# B&R Automation Studio project VisionSample (part 9)

#### Main.st
```iecst
// -----------------------------------------------------------------------------------------------------------
// Use this task to add your own code
// -----------------------------------------------------------------------------------------------------------

// -----------------------------------------------------------------------------------------------------------
// Initialization
// -----------------------------------------------------------------------------------------------------------
PROGRAM _INIT
	cmdLoadRecipeAfterBoot	:= TRUE;
END_PROGRAM

// -----------------------------------------------------------------------------------------------------------
// Cyclic part
// -----------------------------------------------------------------------------------------------------------
PROGRAM _CYCLIC
		// -----------------------------------------------------------------------------------------------------------
	// Vision sensor configuration
	// -----------------------------------------------------------------------------------------------------------
	gVisionImage.CFG.EthDevice				:= 'IF2';			// Ethernet interface for the PLC, this is the IF where you go online
	// Configuration for blob
	gVisionSensor[1].CFG.VisionFunction		:= enumBlob;		// Used to run specific code for this vision function
	gVisionSensor[1].CFG.PowerlinkNode		:= 1;				// Powerlink node number
	gVisionSensor[1].CFG.DataStructure		:= ADR(gBlob);		// Global structures that holds all data related to this function
	gVisionSensor[1].CFG.ComponentLink		:= gCameraBlob;		// Vision component name defined under mappVision in the configuration view
	gVisionSensor[1].CFG.ResolutionWidth_X	:= 1280;
	gVisionSensor[1].CFG.ResolutionHeight_Y	:= 1024;
	// Configuration for code reader
	gVisionSensor[2].CFG.VisionFunction		:= enumCoderReader;
	gVisionSensor[2].CFG.PowerlinkNode		:= 2;
	gVisionSensor[2].CFG.DataStructure		:= ADR(gCodeReader);
	gVisionSensor[2].CFG.ComponentLink		:= gCameraCodeReading;
	gVisionSensor[2].CFG.ResolutionWidth_X	:= 1280;
	gVisionSensor[2].CFG.ResolutionHeight_Y	:= 1024;
	// Configuration for match
	gVisionSensor[3].CFG.VisionFunction		:= enumMatch;
	gVisionSensor[3].CFG.PowerlinkNode		:= 3;
	gVisionSensor[3].CFG.DataStructure		:= ADR(gMatch);
	gVisionSensor[3].CFG.ComponentLink		:= gCameraMatch;
	gVisionSensor[3].CFG.ResolutionWidth_X	:= 1280;
	gVisionSensor[3].CFG.ResolutionHeight_Y	:= 1024;
	// Configuration for meaurement
	gVisionSensor[4].CFG.VisionFunction		:= enumMeasurement;
	gVisionSensor[4].CFG.PowerlinkNode		:= 4;
	gVisionSensor[4].CFG.DataStructure		:= ADR(gMT);
	gVisionSensor[4].CFG.ComponentLink		:= gCameraMeasurement;
	gVisionSensor[4].CFG.ResolutionWidth_X	:= 1280;
	gVisionSensor[4].CFG.ResolutionHeight_Y	:= 1024;
	// Configuration for OCR
	gVisionSensor[5].CFG.VisionFunction		:= enumOCR;
	gVisionSensor[5].CFG.PowerlinkNode		:= 5;
	gVisionSensor[5].CFG.DataStructure		:= ADR(gOCR);
	gVisionSensor[5].CFG.ComponentLink		:= gCameraOCR;
	gVisionSensor[5].CFG.ResolutionWidth_X	:= 1280;
	gVisionSensor[5].CFG.ResolutionHeight_Y	:= 1024;
	// Configuration for PixelCounter
	gVisionSensor[6].CFG.VisionFunction		:= enumPixelCounter;
	gVisionSensor[6].CFG.PowerlinkNode		:= 6;
	gVisionSensor[6].CFG.DataStructure		:= ADR(gPixel);
	gVisionSensor[6].CFG.ComponentLink		:= gCameraPxl;
	gVisionSensor[6].CFG.ResolutionWidth_X	:= 1280;
	gVisionSensor[6].CFG.ResolutionHeight_Y	:= 1024;

	// -----------------------------------------------------------------------------------------------------------
	// Lights configuration
	// -----------------------------------------------------------------------------------------------------------
	// Configuration for backlights
	gVisionLight[1].CFG.LightType		:= enumBacklight;
	gVisionLight[1].CFG.PowerlinkNode	:= 10;
	gVisionLight[1].DAT.FlashColor		:= 1;
	gVisionLight[2].CFG.LightType		:= enumBacklight;
	gVisionLight[2].CFG.PowerlinkNode	:= 11;
	gVisionLight[2].DAT.FlashColor		:= 1;
	// Configuration for lightbars
	gVisionLight[3].CFG.LightType		:= enumLightbar;
	gVisionLight[3].CFG.PowerlinkNode	:= 20;
	gVisionLight[3].DAT.FlashColor		:= 1;

	// -----------------------------------------------------------------------------------------------------------
	// Backlight handling, this block can be deleted when no backlights are used
	// -----------------------------------------------------------------------------------------------------------

	// -----------------------------------------------------------------------------------------------------------
	// Trigger selected backlight when selected sensor is triggered
	IF(EDGEPOS(gVisionSensor[gSelectedSensor].CMD.ImageTrigger)) THEN
		gVisionLight[gSelectedLight].DAT.Exposure		:= gVisionSensor[gSelectedSensor].DAT.Exposure;
		gVisionLight[gSelectedLight].DAT.NettimeDelay	:= gVisionSensor[gSelectedSensor].DAT.NettimeDelay;
		gVisionLight[gSelectedLight].CMD.FlashTrigger	:= TRUE;
	END_IF

	// -----------------------------------------------------------------------------------------------------------
	// Recipe handling, this block can be deleted when no recipes are used
	// -----------------------------------------------------------------------------------------------------------

	// -----------------------------------------------------------------------------------------------------------
	// Transfer data when loading a recipe
	IF EDGENEG(Recipe_01.CMD.Load) OR cmdLoadRecipeAfterBoot THEN
		cmdLoadRecipeAfterBoot := FALSE;
		FOR i := 1 TO MAX_NUM_CAMS DO
			gVisionSensor[i].FCT.ApplicationName	:= RecipeData.Cam[i].ApplicationName;
			gVisionSensor[i].DAT.Exposure			:= RecipeData.Cam[i].Exposure;
			gVisionSensor[i].DAT.FlashColor			:= RecipeData.Cam[i].FlashColor;
			gVisionSensor[i].DAT.FlashSegment		:= RecipeData.Cam[i].FlashSegment;
			gVisionSensor[i].DAT.Focus				:= RecipeData.Cam[i].Focus;
			gVisionSensor[i].DAT.Gain				:= RecipeData.Cam[i].Gain;
			gVisionSensor[i].DAT.MaxItemCnt			:= RecipeData.Cam[i].MaxItemCnt;
			gVisionSensor[i].DAT.Timeout			:= RecipeData.Cam[i].Timeout;
		END_FOR
		FOR i := 1 TO MAX_NUM_LIGHTS DO
			gVisionLight[i].DAT.Exposure			:= RecipeData.Light[i].Exposure;
			gVisionLight[i].DAT.FlashColor			:= RecipeData.Light[i].FlashColor;
			gVisionLight[i].DAT.FlashSegment		:= RecipeData.Light[i].FlashSegment;
			gVisionLight[i].DAT.SetAngle			:= RecipeData.Light[i].SetAngle;
			gVisionLight[i].DAT.Timeout				:= RecipeData.Light[i].Timeout;
		END_FOR
		// Switch vision application when recipe for blob was loaded
		gVisionSensor[1].CMD.VaSwitchApplication := TRUE;
	END_IF

	// -----------------------------------------------------------------------------------------------------------
	// Transfer data cyclic to the remanent variable
	IF NOT Recipe_01.CMD.Load THEN
		FOR i := 1 TO MAX_NUM_CAMS DO
			RecipeData.Cam[i].ApplicationName	:= gVisionSensor[i].FCT.ApplicationName;
			RecipeData.Cam[i].Exposure			:= gVisionSensor[i].DAT.Exposure;
			RecipeData.Cam[i].FlashColor		:= gVisionSensor[i].DAT.FlashColor;
			RecipeData.Cam[i].FlashSegment		:= gVisionSensor[i].DAT.FlashSegment;
			RecipeData.Cam[i].Focus				:= gVisionSensor[i].DAT.Focus;
			RecipeData.Cam[i].Gain				:= gVisionSensor[i].DAT.Gain;
			RecipeData.Cam[i].MaxItemCnt		:= gVisionSensor[i].DAT.MaxItemCnt;
			RecipeData.Cam[i].Timeout			:= gVisionSensor[i].DAT.Timeout;
		END_FOR
		FOR i := 1 TO MAX_NUM_LIGHTS DO
			RecipeData.Light[i].Exposure		:= gVisionLight[i].DAT.Exposure;
			RecipeData.Light[i].FlashColor		:= gVisionLight[i].DAT.FlashColor;
			RecipeData.Light[i].FlashSegment	:= gVisionLight[i].DAT.FlashSegment;
			RecipeData.Light[i].SetAngle		:= gVisionLight[i].DAT.SetAngle;
			RecipeData.Light[i].Timeout			:= gVisionLight[i].DAT.Timeout;
		END_FOR
	END_IF
	IF visSaveRecipe OR visNewRecipe THEN
		IF(visNewRecipe) THEN
			Recipe_01.CMD.New := TRUE;
		ELSE
			Recipe_01.CMD.Save := TRUE;
		END_IF
		visNewRecipe := FALSE;
		visSaveRecipe := FALSE;
	END_IF
END_PROGRAM
```

### Package Logical/Programs/Axis - Program that handles motion axis related tasks

### Program Logical/Programs/Axis/Axis

#### Types.typ
```iecst
TYPE
	hmi_out_typ : 	STRUCT
		positon : REAL;
		veleocity : REAL;
		inVelocity : BOOL;
		inPostion : BOOL;
		powerlinkCycle_us : DINT;
		triggerPosDelta : REAL;
		triggerTimeDelta : DINT; (*In us*)
	END_STRUCT;
	recipe_typ : 	STRUCT
		acceleration : REAL := 360;
		velocity : REAL := 36000;
		axisPositionDelayCycles : REAL;
		visionPreTriggerCycles : REAL;
		axisPositionTrigger : REAL;
		axisPeriod : REAL;
	END_STRUCT;
	hmi_in_cmd_typ : 	STRUCT
		moveAbs : BOOL;
		home : BOOL;
		power : BOOL;
		run : BOOL;
		errReset : BOOL;
	END_STRUCT;
	hmi_in_typ : 	STRUCT
		recipe : recipe_typ;
		cmd : hmi_in_cmd_typ;
	END_STRUCT;
	hmi_typ : 	STRUCT
		in : hmi_in_typ;
		out : hmi_out_typ;
	END_STRUCT;
	local_typ : 	STRUCT
		mpAxisBasic_0 : MpAxisBasic;
		mpAxisBasicPar_0 : MpAxisBasicParType;
		nettimeLastCycle_us : DINT;
		powerlinkCycle_us : DINT;
		axisPositionNow : REAL;
		triggerPosDelta : REAL;
		triggerTimeDelta : DINT; (*In us*)
		mpRecipeRegVar : MpRecipeRegParSync;
	END_STRUCT;
	hw_in_typ : 	STRUCT
		nettime : DINT;
	END_STRUCT;
	hw_typ : 	STRUCT
		in : hw_in_typ;
	END_STRUCT;
END_TYPE
```

#### Main.st
```iecst
// --------------------------------------------------------------------------------------------------------------------
// Motion sample for using nettime
// --------------------------------------------------------------------------------------------------------------------
PROGRAM _INIT
	this.mpAxisBasic_0.Enable			:= TRUE;
	this.mpAxisBasic_0.MpLink			:= ADR(gAxis_1);
	this.mpAxisBasic_0.Parameters		:= ADR(this.mpAxisBasicPar_0);
	this.mpAxisBasic_0();
	this.mpAxisBasicPar_0.Homing.Mode	:= mcHOMING_DEFAULT;

	hmi.in.recipe.axisPeriod				:= 360; // Needs also to be set in the axis configuration
	hmi.in.recipe.axisPositionTrigger		:= 0;
	hmi.in.recipe.axisPositionDelayCycles	:= 1; 	// Number of PLK cycles which the axis position is old when it comes to this task (Time from encoder to now in this task)
	hmi.in.recipe.visionPreTriggerCycles	:= 4; 	// Number of powerlink cycles the trigger has to be send ahead
	// For camera only 4 is good value, for backlight use 12 with a 800us Powerlink cylce

END_PROGRAM

// -----------------------------------------------------------------------------------------------------------
// Cyclic part
// -----------------------------------------------------------------------------------------------------------
PROGRAM _CYCLIC

// -----------------------------------------------------------------------------------------------------------
// Mapp Motion Axis control
// -----------------------------------------------------------------------------------------------------------
	this.mpAxisBasic_0.Power				:= this.mpAxisBasic_0.Active AND this.mpAxisBasic_0.Info.ReadyToPowerOn AND hmi.in.cmd.power;
	this.mpAxisBasic_0.ErrorReset			:= hmi.in.cmd.errReset;
	this.mpAxisBasic_0.Home					:= this.mpAxisBasic_0.PowerOn AND NOT this.mpAxisBasic_0.IsHomed XOR hmi.in.cmd.home;
	this.mpAxisBasic_0.MoveVelocity			:= this.mpAxisBasic_0.PowerOn AND this.mpAxisBasic_0.IsHomed AND hmi.in.cmd.run;

	IF this.mpAxisBasic_0.PowerOn AND this.mpAxisBasic_0.IsHomed AND hmi.in.cmd.moveAbs THEN
		this.mpAxisBasic_0.MoveAbsolute		:= TRUE;
		this.mpAxisBasicPar_0.Position		:= hmi.in.recipe.axisPositionTrigger;
	END_IF
	hmi.in.cmd.moveAbs					:= FALSE;

	IF hmi.in.recipe.velocity <> this.mpAxisBasicPar_0.Velocity OR hmi.in.recipe.acceleration <> this.mpAxisBasicPar_0.Acceleration THEN
		this.mpAxisBasicPar_0.Velocity		:= hmi.in.recipe.velocity;
		this.mpAxisBasicPar_0.Acceleration	:= hmi.in.recipe.acceleration;
		this.mpAxisBasicPar_0.Deceleration	:= hmi.in.recipe.acceleration;
		this.mpAxisBasic_0.Update			:= TRUE;
	END_IF

	this.mpAxisBasic_0();

	IF hw.in.nettime > this.nettimeLastCycle_us THEN
		this.powerlinkCycle_us	:= hw.in.nettime - this.nettimeLastCycle_us;
	ELSE
		this.powerlinkCycle_us	:= -2147483648-hw.in.nettime + 2147483647-this.nettimeLastCycle_us; // handle wrap around
	END_IF
	this.nettimeLastCycle_us		:= hw.in.nettime;

	hmi.out.inVelocity 	:= gAxis.status.inVelocity	:= 	this.mpAxisBasic_0.InVelocity;
	hmi.out.veleocity 	:= gAxis.status.velocity	:= 	this.mpAxisBasic_0.Velocity;
	hmi.out.inPostion 								:=	this.mpAxisBasic_0.InPosition;
	// When the MpAxis gives us the read position, it is old. So calculate the "now" position
	hmi.out.positon 	:= gAxis.status.position	:= 	LREAL_TO_REAL(this.mpAxisBasic_0.Position) + this.mpAxisBasic_0.Velocity * DINT_TO_REAL(this.powerlinkCycle_us) * hmi.in.recipe.axisPositionDelayCycles / 1000000; ;

	IF this.mpAxisBasic_0.UpdateDone THEN
		this.mpAxisBasic_0.Update := FALSE;
	END_IF

	IF this.mpAxisBasic_0.InPosition THEN
		this.mpAxisBasic_0.MoveAbsolute		:= FALSE;
	END_IF

	// -----------------------------------------------------------------------------------------------------------
	// Calulate time to camera trigger point
	// -----------------------------------------------------------------------------------------------------------

	// calculate axis postion in the current period
	IF this.axisPositionNow > hmi.in.recipe.axisPeriod THEN // modulo correction
		this.axisPositionNow		:= hmi.out.positon- hmi.in.recipe.axisPeriod;
	ELSIF this.axisPositionNow < 0 THEN // modulo correction
		this.axisPositionNow		:= hmi.out.positon + hmi.in.recipe.axisPeriod;
	END_IF

	// calculate differen (triggerPosDelta) in current axis postion to the trigger postion
	IF this.mpAxisBasic_0.Velocity > 0 THEN
		this.triggerPosDelta		:= hmi.in.recipe.axisPositionTrigger - this.axisPositionNow;
	ELSE
		this.triggerPosDelta		:= this.axisPositionNow - hmi.in.recipe.axisPositionTrigger;
	END_IF

	IF this.triggerPosDelta < 0 THEN // modulo correction
		this.triggerPosDelta		:= this.triggerPosDelta + hmi.in.recipe.axisPositionTrigger;
	END_IF

	IF hmi.out.veleocity > 0 THEN
		// convert position difference to a time difference (the time until the axis is at the trigger postion with the current velocity)
		gAxis.status.triggerTimeDelta 	:= LREAL_TO_DINT((this.triggerPosDelta / this.mpAxisBasic_0.Velocity) * 1000000);
	END_IF

	gAxis.status.nettime 		  		:= hw.in.nettime;
	gAxis.status.powerlinkCycleTime 	:= this.powerlinkCycle_us;

	hmi.out.triggerPosDelta 	:= this.triggerPosDelta;
	hmi.out.powerlinkCycle_us 	:= this.powerlinkCycle_us;
	hmi.out.triggerTimeDelta 	:= this.triggerTimeDelta;

	this.mpRecipeRegVar.Enable 		:= gRecipe.out.active;
	this.mpRecipeRegVar.MpLink 		:= gRecipe.out.mpLink;
	this.mpRecipeRegVar.ConfirmSave := this.mpRecipeRegVar.SaveNotification;
	this.mpRecipeRegVar.Category 	:= ADR('Recipe');
	this.mpRecipeRegVar.PVName 		:= ADR('::Axis:hmi.in.recipe');
	this.mpRecipeRegVar();

	// Clear ready for init (auto load) if data structures have not been registred
	IF NOT this.mpRecipeRegVar.Active THEN
		gRecipe.in.readyForInit := FALSE;
	END_IF

END_PROGRAM
```

### Package Logical/Programs/Files - Program that handles file system tasks

### gFiles.typ
```iecst
TYPE
	gFiles_input_typ : 	STRUCT
		refresh : BOOL;
	END_STRUCT;
	gFiles_output_typ : 	STRUCT
		fileDevice : STRING[10];
		ready : BOOL;
	END_STRUCT;
	gFiles_typ : 	STRUCT
		output : gFiles_output_typ;
		input : gFiles_input_typ;
	END_STRUCT;
END_TYPE
```

### Program Logical/Programs/Files/Files

#### Types.typ
```iecst
TYPE
	local_typ : 	STRUCT
		brdkFileDevUsb : brdkFileDeviceHandler;
		brdkFileDev : brdkFileDeviceHandler;
		mpFileManUI : MpFileManagerUI;
		mpFileUISetup : MpFileManagerUISetupType;
		mappView : brdkViImg_mappView;
		lastFileName : STRING[255];
		brdkFileRead : brdkFileRead;
		fileName : STRING[255];
		fileType : STRING[5];
		delayTon : TON;
		setIdx : BOOL;
	END_STRUCT;
	hmi_in_cmd_typ : 	STRUCT
		deleteAllImages : BOOL;
		selectedIdx : UINT;
		download : BOOL;
	END_STRUCT;
	hmi_in_typ : 	STRUCT
		cmd : hmi_in_cmd_typ;
	END_STRUCT;
	hmi_out_typ : 	STRUCT
		enableDeleteAllImageBtn : BOOL;
		fileNames : ARRAY[0..FILES_LIST_SIZE]OF STRING[255];
		loadFileStatus : STRING[200];
		img : STRING[8000000];
		svg : STRING[1000000];
		downloadSrc : STRING[500];
	END_STRUCT;
	hmi_typ : 	STRUCT
		in : hmi_in_typ;
		out : hmi_out_typ;
		mpFile : MpFileManagerUIConnectType;
	END_STRUCT;
END_TYPE
```

#### Variables.var
```iecst
VAR CONSTANT
	FILES_LIST_SIZE : USINT := 13; (*Number of files to be displayed on one page of the list in the HMI application*)
END_VAR
VAR
	hmi : hmi_typ;
	i : UINT;
	this : local_typ;
END_VAR
```

#### Main.st
```iecst
PROGRAM _INIT
	(* Insert code here *)
	this.brdkFileDev.enable := TRUE;
	this.brdkFileDev.setup.plcDrive := F_DRIVE;
	this.brdkFileDev.setup.usbOverrule := FALSE;
	this.brdkFileDev.simulation.pcRootFolder := 'plcSim\MappVisionDemo';
	this.brdkFileDev.simulation.pcHDDrive := C_DRIVE;
	this.brdkFileDev.setup.rootFileDeviceName := 'ROOT_PLC';

	this.brdkFileDev.setup.fileDevices[0].name := 'SIM_BLOB';
	this.brdkFileDev.setup.fileDevices[0].path := 'sim/BLOB';
	this.brdkFileDev.setup.fileDevices[1].name := 'SIM_CR';
	this.brdkFileDev.setup.fileDevices[1].path := 'sim/CR';
	this.brdkFileDev.setup.fileDevices[2].name := 'SIM_MATCH';
	this.brdkFileDev.setup.fileDevices[2].path := 'sim/Match';
	this.brdkFileDev.setup.fileDevices[3].name := 'SIM_MEAS';
	this.brdkFileDev.setup.fileDevices[3].path := 'sim/Measurement';
	this.brdkFileDev.setup.fileDevices[4].name := 'SIM_OCR';
	this.brdkFileDev.setup.fileDevices[4].path := 'sim/OCR';
	this.brdkFileDev.setup.fileDevices[5].name := 'SIM_PXCNT';
	this.brdkFileDev.setup.fileDevices[5].path := 'sim/PxCnt';

	this.brdkFileDevUsb.setup.plcDrive := F_DRIVE;
	this.brdkFileDevUsb.setup.usbOverrule := TRUE;
	this.brdkFileDevUsb.simulation.pcRootFolder := 'plcSim\MappVisionDemo';
	this.brdkFileDevUsb.simulation.pcHDDrive := C_DRIVE;
	this.brdkFileDevUsb.simulation.pcUSBDrive := D_DRIVE;
	this.brdkFileDevUsb.setup.rootFileDeviceName := 'ROOT_USB';

	this.brdkFileDevUsb.setup.fileDevices[0].name := 'IMG';
	this.brdkFileDevUsb.setup.fileDevices[0].path := 'images';
	this.brdkFileDevUsb.setup.fileDevices[1].name := 'RECIPE';
	this.brdkFileDevUsb.setup.fileDevices[1].path := 'Recipe';
	this.brdkFileDevUsb.setup.fileDevices[2].name := 'VI_DIAG';
	this.brdkFileDevUsb.setup.fileDevices[2].path := 'visionDiag';
	this.brdkFileDevUsb.setup.fileDevices[3].name := 'DATA';
	this.brdkFileDevUsb.setup.fileDevices[3].path := 'data';

	this.mpFileManUI.UISetup.FileListScrollWindow := 1;
	this.mpFileManUI.UISetup.FileListSize := FILES_LIST_SIZE;

	this.mappView.simulateConfig.activate := TRUE;
	this.mappView.simulateConfig.appendNumber := FALSE;
	this.mappView.simulateConfig.autoIncrementNumber := FALSE;
	this.mappView.simulateConfig.pDevice := ADR('IMG');
	this.mappView.simulateConfig.useRandomNumbers := FALSE;

	hmi.mpFile.File.Filter := '*jpg';

END_PROGRAM

PROGRAM _CYCLIC
	(* Insert code here *)

	// Create file devices
	this.brdkFileDev();

	IF EDGEPOS(this.brdkFileDev.ready) THEN
		this.brdkFileDevUsb.enable := TRUE;
	END_IF

	hmi.mpFile.File.Refresh := hmi.mpFile.File.Refresh OR gFiles.input.refresh;
	gFiles.input.refresh := FALSE;
	this.brdkFileDevUsb();

	gFiles.output.fileDevice := 'ROOT';
	gFiles.output.ready := this.brdkFileDevUsb.ready;

	// Use MpFile to handle the images files
	hmi.mpFile.DeviceList.DeviceNames[0] := 'IMG';

	this.mpFileManUI.Enable := this.brdkFileDevUsb.ready;
	this.mpFileManUI.MpLink := ADR(gFileManagerUI);
	this.mpFileManUI.UIConnect := ADR(hmi.mpFile);
	IF hmi.mpFile.File.List.PageDown OR hmi.mpFile.File.List.PageUp OR hmi.mpFile.File.List.StepDown OR hmi.mpFile.File.List.StepUp THEN
		this.setIdx := TRUE;
	END_IF

	IF NOT hmi.mpFile.File.List.Items[hmi.in.cmd.selectedIdx].IsSelected THEN
		IF this.setIdx THEN
			this.setIdx := FALSE;
		ELSE

			FOR i := 0 TO this.mpFileManUI.UISetup.FileListSize BY 1 DO
				hmi.mpFile.File.List.Items[i].IsSelected := i = hmi.in.cmd.selectedIdx;
			END_FOR
		END_IF

	END_IF

	this.mpFileManUI();

	FOR i:= 0 TO this.mpFileManUI.UISetup.FileListSize BY 1 DO
		hmi.out.fileNames[i] := hmi.mpFile.File.List.Items[i].Name;
	END_FOR

	IF this.setIdx THEN
		FOR i := 0 TO this.mpFileManUI.UISetup.FileListSize BY 1 DO
			IF hmi.mpFile.File.List.Items[i].IsSelected THEN
				hmi.in.cmd.selectedIdx := i;
			END_IF
		END_FOR
	END_IF

	// Load image and overlay when the selected image changes.
	IF hmi.mpFile.File.List.Items[hmi.in.cmd.selectedIdx].Name <> this.lastFileName THEN
		this.fileName := hmi.mpFile.File.List.Items[hmi.in.cmd.selectedIdx].Name;
		brsstrcpy(ADR(this.fileType),ADR(this.fileName)+brsstrlen(ADR(this.fileName))-3);

		brsstrcpy(ADR(this.fileName)+brsstrlen(ADR(this.fileName))-4,ADR(''));
		this.mappView.simulateConfig.pFile := ADR(this.fileName);

		IF this.fileType = 'jpg' THEN
			this.mappView.imageFormat := BRDKVIIMG_IMG_TYPE_JPEG;
		ELSE
			this.mappView.imageFormat := BRDKVIIMG_IMG_TYPE_BMP;
		END_IF

		this.mappView.updateImage := TRUE;
		this.brdkFileRead.enable := TRUE;

		this.brdkFileRead.fileDevice := hmi.mpFile.DeviceList.DeviceNames[hmi.mpFile.DeviceList.SelectedIndex];
		this.brdkFileRead.fileName := hmi.mpFile.File.List.Items[hmi.in.cmd.selectedIdx].Name;
		brsstrcpy(ADR(this.brdkFileRead.fileName)+brsstrlen(ADR(this.brdkFileRead.fileName))-3,ADR('svg'));
		this.brdkFileRead.pData := ADR(hmi.out.svg);
		this.brdkFileRead.dataLength := SIZEOF(hmi.out.svg);

	END_IF

	this.lastFileName := hmi.mpFile.File.List.Items[hmi.in.cmd.selectedIdx].Name;
	this.brdkFileRead();

	IF this.brdkFileRead.done OR this.brdkFileRead.status = fiERR_FILE_NOT_FOUND THEN
		this.brdkFileRead.enable := FALSE;
	END_IF

	IF hmi.mpFile.MessageBox.Type =  mpFILE_MSG_CONFIRM_DELETE THEN
		hmi.mpFile.MessageBox.Confirm := TRUE;
	END_IF

	IF hmi.in.cmd.download THEN
		hmi.in.cmd.download	:= FALSE;
		this.delayTon.IN 	:= TRUE;
		this.delayTon.PT 	:= T#400ms;

		hmi.out.downloadSrc := '<script>function onSvgLoad() {const link = document.createElement("a");link.href = "/FileDevice:';
		brsstrcat(ADR(hmi.out.downloadSrc),ADR(this.brdkFileRead.fileDevice));
		brsstrcat(ADR(hmi.out.downloadSrc),ADR('/'));
		brsstrcat(ADR(hmi.out.downloadSrc),ADR(hmi.mpFile.File.List.Items[hmi.in.cmd.selectedIdx].Name));
		brsstrcat(ADR(hmi.out.downloadSrc),ADR('";link.download="'));
		brsstrcat(ADR(hmi.out.downloadSrc),ADR(hmi.mpFile.File.List.Items[hmi.in.cmd.selectedIdx].Name));
		brsstrcat(ADR(hmi.out.downloadSrc),ADR('";link.click();}; onSvgLoad(); </script>'));
	END_IF

	IF this.delayTon.Q THEN
		this.delayTon.IN := FALSE;
		hmi.out.downloadSrc := '';
	END_IF
	this.delayTon();

	hmi.out.loadFileStatus := this.brdkFileRead.description;

	this.mappView.enable := this.brdkFileDevUsb.ready;
	this.mappView.wsPort :=  18100;
	//	this.mappView.pSvgImage := ADR(hmi.out.img);
	//	this.mappView.maxSvgImageLength := SIZEOF(hmi.out.img);
	this.mappView();

END_PROGRAM

PROGRAM _EXIT
	(* Insert code here *)
	this.brdkFileDev(	enable := FALSE);
	this.brdkFileDevUsb(enable := FALSE);
	this.mappView(		enable := FALSE);
	this.mpFileManUI(	Enable := FALSE);

END_PROGRAM
```

### Package Logical/Programs/Vision - Main program that handles triggering and processing of vision

### Program Logical/Programs/Vision/Vision (IEC)

#### Main.st - Init, cyclic, exit code
```iecst
// --------------------------------------------------------------------------------------------------------------------
// General vision task. This is a support task for the mappVision. The following functions are implemneted
// - Translate some values in text messages
// - Reset camera trigger when inspection is finsihed
// - Load vision application
// - Save diagnostic data
// Version 2.x (Check revision history for details)
// --------------------------------------------------------------------------------------------------------------------
PROGRAM _INIT

	userInitCommonPreAction;

	FOR idx:= START_IDX TO MAX_NUM_CAMS BY 1 DO
		setupPointersAction;

		//  Create IO path to cam
		this.path := 'IF3.ST';
		tmpStr := USINT_TO_STRING(idx);
		brsstrcat(ADR(this.path),ADR(tmpStr));

		this.recipePVName := '::Vision1:hmiInstance[';
		brsstrcat(ADR(this.recipePVName),ADR(tmpStr));
		brsstrcat(ADR(this.recipePVName),ADR('].in.recipe'));

		// Create IO path to lights
		FOR i := START_IDX TO MAX_NUM_LIGHTS BY 1 DO
			this.lightPath[i] := 'IF3.ST';
			tmpStr := USINT_TO_STRING(idx*16+(i-1));
			brsstrcat(ADR(this.lightPath[i]),ADR(tmpStr));
		END_FOR

		FOR i:= START_IDX TO MAX_NUM_RESULTS BY 1 DO
			hmi.out.tableVF.tableNum[i] := i;
		END_FOR

		hmi.out.wsPort := 18000+idx*10;
		this.mappView.enable := TRUE;
		this.mappView.wsPort := hmi.out.wsPort;
		this.mappView.simulateConfig.activate := DiagCpuIsSimulated();
		this.mappView.simulateConfig.pFile := ADR('img');
		this.mappView.simulateConfig.useRandomNumbers := FALSE;
		this.mappView.simulateConfig.appendNumber := TRUE;
		this.mappView.simulateConfig.autoIncrementNumber := TRUE;
		this.mappView.simulateConfig.minNumber := 1;
		this.mappView.simulateConfig.maxNumber := 3;

		this.visionDiagFileDevice := 'VI_DIAG'; // File device is created in Files program (changes to USB if such is pluged in)

		hmi.out.camera.plNodeNr := idx;
		hmi.in.recipe.cam.focus := 200;
		hmi.in.recipe.cam.exposureTime := 100;

		hmi.in.cmd.resetInfo := TRUE;

		// -----------------------------------------------------------------------------------------------------------
		// Set camera specific data
		// -----------------------------------------------------------------------------------------------------------

		hmi.in.cmd.resultTabIndex := 5;
		CASE idx OF
			1:
				this.mappView.pMappLink := ADR(gCameraBlob);
				this.mappView.simulateConfig.pDevice := ADR('SIM_BLOB');
				hmi.out.camera.visionFunction := 'BLOB';
				hmi.out.usedVF.BLOB := TRUE;
				hmi.in.cmd.resultTabIndex := MIN(hmi.in.cmd.resultTabIndex,idx-1);
			2:
				this.mappView.pMappLink := ADR(gCameraCodeReading);
				this.mappView.simulateConfig.pDevice := ADR('SIM_CR');
				hmi.out.camera.visionFunction := 'Code Reader';
				hmi.out.usedVF.codeReader := TRUE;
				hmi.in.cmd.resultTabIndex := MIN(hmi.in.cmd.resultTabIndex,idx-1);
				(*hmi.out.VF.numResults*)
			3:
				this.mappView.pMappLink := ADR(gCameraMatch);
				this.mappView.simulateConfig.pDevice := ADR('SIM_MATCH');
				hmi.out.camera.visionFunction := 'Matching';
				hmi.out.usedVF.matching := TRUE;
				hmi.in.cmd.resultTabIndex := MIN(hmi.in.cmd.resultTabIndex,idx-1);
			4:
				this.mappView.pMappLink := ADR(gCameraMeasurement);
				this.mappView.simulateConfig.pDevice := ADR('SIM_MEAS');
				hmi.out.camera.visionFunction := 'Measurement';
				hmi.out.usedVF.measurement := TRUE;
				hmi.in.cmd.resultTabIndex := MIN(hmi.in.cmd.resultTabIndex,idx-1);
			5:
				this.mappView.pMappLink := ADR(gCameraOCR);
				this.mappView.simulateConfig.pDevice := ADR('SIM_OCR');
				hmi.out.camera.visionFunction := 'OCR';
				hmi.out.usedVF.OCR := TRUE;
				hmi.in.cmd.resultTabIndex := MIN(hmi.in.cmd.resultTabIndex,idx-1);
			6:
				this.mappView.pMappLink := ADR(gCameraPxl);
				this.mappView.simulateConfig.pDevice := ADR('SIM_PXCNT');
				hmi.out.camera.visionFunction := 'Pixel Counter';
				hmi.out.usedVF.pixelCounter := TRUE;
				hmi.in.cmd.resultTabIndex := MIN(hmi.in.cmd.resultTabIndex,idx-1);

		END_CASE

		userInitLocalPostAction;

	END_FOR

END_PROGRAM

// -----------------------------------------------------------------------------------------------------------
// Cyclic part
// -----------------------------------------------------------------------------------------------------------
PROGRAM _CYCLIC

	userCommonPreAction; // user common action before all other

	FOR idx:= START_IDX TO MAX_NUM_CAMS BY 1 DO
		setupPointersAction;

		userLocalPreAction; // user local action before all other

		// -----------------------------------------------------------------------------------------------------------
		// Translate camera status in readable text
		// -----------------------------------------------------------------------------------------------------------
		IF hw.camera.in.common.moduleOk THEN
			brdkViBase_camStatusToString(hw.camera.in.status.cameraStatus,ADR(hmi.out.camera.statusText));
		ELSE
			hmi.out.camera.statusText := 'Disconnected';
		END_IF

		// -----------------------------------------------------------------------------------------------------------
		// Check if vision cockpit is open
		// -----------------------------------------------------------------------------------------------------------
		hmi.out.camera.mappVisionActive := (hw.camera.in.status.cameraStatus AND 16#8000_0000) > 0;

		// -----------------------------------------------------------------------------------------------------------
		// Read camera hardware info
		// -----------------------------------------------------------------------------------------------------------

		IF hmi.in.cmd.resetInfo THEN
			hmi.in.cmd.resetInfo := FALSE;
			hmi.in.cameraInfo.distance := hmi.in.recipe.cam.focus;
			this.brdkViBase_getCameraInfo_0.execute := TRUE;
			this.brdkViBase_getCameraInfo_0.pluggedModule := hw.camera.in.common.moduleOk AND NOT DiagCpuIsSimulated();

			FOR i := START_IDX TO MAX_NUM_LIGHTS BY 1 DO
				this.brdkViBase_getLightInfo[i].execute := TRUE;
				this.brdkViBase_getLightInfo[i].pInfo := ADR(hmi.out.lights[i].info);
				this.brdkViBase_getLightInfo[i].pDevicePath := ADR(this.lightPath[i]);
				this.brdkViBase_getLightInfo[i].pluggedModule := hw.lights[i].in.common.moduleOk AND NOT DiagCpuIsSimulated();
			END_FOR

		END_IF

		this.brdkViBase_getCameraInfo_0.pDevicePath := ADR(this.path);
		this.brdkViBase_getCameraInfo_0.pInfo := ADR(hmi.in.cameraInfo);
		this.brdkViBase_getCameraInfo_0();

		FOR i:=START_IDX TO MAX_NUM_LIGHTS BY 1 DO
			this.brdkViBase_getLightInfo[i]();

			IF hmi.out.lights[i].info.orderNr <> '' AND this.brdkViBase_getLightInfo[i].status = ERR_OK THEN
				// set Camera flash options based on current camera
				brdkViBase_LEDColorToOptions(hmi.out.lights[i].info.LED_color, ADR(hmi.out.lights[i].flashLightOptions));
			END_IF
		END_FOR

		IF hw.camera.out.par.focus <> hmi.in.recipe.cam.focus THEN
			hmi.in.cameraInfo.distance := hmi.in.recipe.cam.focus;
		END_IF

		IF hmi.in.cameraInfo.orderNr <> '' AND this.brdkViBase_getCameraInfo_0.status = ERR_OK THEN
			brdkViBase_calcOpticInfo(hmi.in.cameraInfo, hmi.out.camera.opticInfo); // calculate optic info based on defined info

			// set Camera flash options based on current camera
			brdkViBase_LEDColorToOptions(hmi.in.cameraInfo.LED_color, ADR(hmi.out.camera.flashLightOptions));
		END_IF

		IF hw.io.in.nettime > this.axisTrig.nettimeLastCycle_us THEN
			this.axisTrig.powerlinkCycle_us	:= hw.io.in.nettime - this.axisTrig.nettimeLastCycle_us;
		ELSE
			this.axisTrig.powerlinkCycle_us	:= -2147483648-hw.io.in.nettime + 2147483647-this.axisTrig.nettimeLastCycle_us; // handle wrap around
		END_IF
		this.axisTrig.nettimeLastCycle_us	:= hw.io.in.nettime;

		// -----------------------------------------------------------------------------------------------------------
		// Image trigger (camera and lights)
		// -----------------------------------------------------------------------------------------------------------
		hmi.in.recipe.cam.flashColor := STRING_TO_USINT(hmi.in.recipe.cam.flashColorStr);
		hw.camera.out.par.focus 			:= hmi.in.recipe.cam.focus;
		hw.camera.out.par.flashSegment	 	:= hmi.in.recipe.cam.flashSegment;
		hw.camera.out.par.flashColor 		:= hmi.in.recipe.cam.flashColor;
		hw.camera.out.par.exposureTime 		:= hmi.in.recipe.cam.exposureTime;
		hw.camera.out.par.chromaticLock 	:= hmi.in.recipe.cam.chromaticLock;
		hw.camera.out.par.gainLevel 		:= hmi.in.recipe.cam.gainLevel;
		hw.camera.out.par.IRFilter			:= hmi.in.recipe.cam.IRFilter;

		//-------------------------------------------------------------------------

		// Copy recipe data (e.g. enable, maximal number of results, etc.)
		hw.VF.blob.out			:=hmi.in.recipe.BLOB;
		hw.VF.codeReader.out	:= hmi.in.recipe.CR;
		hw.VF.matching.out		:=hmi.in.recipe.match;
		hw.VF.measurement.out	:=hmi.in.recipe.meassurement;
		hw.VF.ocr.out			:=hmi.in.recipe.OCR;
		hw.VF.pixelCnt.out		:=hmi.in.recipe.pxCnt;

		hmi.out.camera.processingTime:=hw.camera.in.status.cameraProcessingTime;

		CASE idx OF
			1:
				hmi.out.VF.processingTime := hw.VF.blob.in.common.functionProcessingTime;
				hmi.out.VF.numResults := hw.VF.blob.in.common.numResults;
			2:
				hmi.out.VF.processingTime := hw.VF.codeReader.in.common.functionProcessingTime;
				hmi.out.VF.numResults := hw.VF.codeReader.in.common.numResults;
			3:
				hmi.out.VF.processingTime := hw.VF.matching.in.common.functionProcessingTime;
				hmi.out.VF.numResults := hw.VF.matching.in.common.numResults;
			4:
				hmi.out.VF.processingTime := hw.VF.measurement.in.common.functionProcessingTime;
				hmi.out.VF.numResults := hw.VF.measurement.in.common.numResults;
			5:
				hmi.out.VF.processingTime := hw.VF.ocr.in.common.functionProcessingTime;
				hmi.out.VF.numResults := hw.VF.ocr.in.common.numResults;
			6:
				hmi.out.VF.processingTime := hw.VF.pixelCnt.in.common.functionProcessingTime;
				hmi.out.VF.numResults := hw.VF.pixelCnt.in.common.numResults;
		END_CASE;

		//-------------------------------------------------------------------------

		this.ioTrigger(CLK := hw.io.in.commonTrigger OR hw.io.in.individualTrigger);
		this.repetitiveTriggerTON.IN := hmi.in.recipe.repetitiveTrigger;
		this.repetitiveTriggerTON.PT := UDINT_TO_TIME(hmi.in.recipe.repetitiveTriggerInterval);
		this.repetitiveTriggerTON();

		// check if camera is ready for an image trigger and MappView have been updated
		IF this.brdkViBase_imgTrigger_0.ready AND NOT this.brdkViBase_imgTrigger_0.busy AND this.mappView.status = 0 THEN

			// Hmi manual trigger
			IF hmi.in.cmd.trigger OR this.repetitiveTriggerTON.Q THEN
				hmi.in.cmd.trigger 							:= FALSE;

				this.repetitiveTriggerTON(IN:=FALSE);

				this.brdkViBase_imgTrigger_0.trigger 		:= TRUE;
				this.brdkViBase_imgTrigger_0.delayNettime 	:= hw.io.in.nettime + gAxis.status.powerlinkCycleTime * 12+10000; // Calc nettime close to currnet time
				this.currentTriggerNum := 1;
				// Axis trigger
			ELSIF hmi.in.recipe.enableAxisTrigger AND
				gAxis.status.triggerTimeDelta >= (commonHmi.in.recipe.visionPreTriggerCycles * this.axisTrig.powerlinkCycle_us) AND
				gAxis.status.triggerTimeDelta <= ((commonHmi.in.recipe.visionPreTriggerCycles + 1) * this.axisTrig.powerlinkCycle_us) THEN

				this.brdkViBase_imgTrigger_0.trigger := TRUE;
				this.brdkViBase_imgTrigger_0.delayNettime := gAxis.status.nettime + gAxis.status.triggerTimeDelta; // Use time calculated in Axis program
			ELSIF hmi.in.recipe.enableIoTrigger AND this.ioTrigger.Q THEN

				this.brdkViBase_imgTrigger_0.trigger := TRUE;
				this.brdkViBase_imgTrigger_0.delayNettime := gAxis.status.nettime + hmi.in.recipe.ioTriggerDelay ; // Use time calculated in Axis program

			ELSIF this.currentTriggerNum < hmi.in.recipe.multiCaptureNum AND NOT hmi.in.recipe.repetitiveTrigger THEN

				this.brdkViBase_imgTrigger_0.trigger 		:= TRUE;
				this.brdkViBase_imgTrigger_0.delayNettime 	:= hw.io.in.nettime + gAxis.status.powerlinkCycleTime * 12+10000; // Calc nettime close to currnet time

				this.currentTriggerNum := 		this.currentTriggerNum +1;

			END_IF
		END_IF

		this.brdkViBase_imgTrigger_0.searchAcquisitonSettings := hmi.in.cmd.autoSearch;
		this.brdkViBase_imgTrigger_0.pCameraHw := ADR(hw.camera);
		this.brdkViBase_imgTrigger_0.numLights := MAX_NUM_LIGHTS;
		this.brdkViBase_imgTrigger_0.pLightHw := ADR(hw.lights);
		this.brdkViBase_imgTrigger_0.useCamColorForLight := hmi.in.recipe.useCamLedColorForLight;
		this.brdkViBase_imgTrigger_0.useCamExpTimeForLight := hmi.in.recipe.useCamExpTimeForLight;
		this.brdkViBase_imgTrigger_0.simulate.enable := DiagCpuIsSimulated();
		this.brdkViBase_imgTrigger_0.simulate.alwaysSimulateNonePresentLights := TRUE;
		this.brdkViBase_imgTrigger_0.simulate.imgProcessingDelay := T#300ms;
		this.brdkViBase_imgTrigger_0();

		FOR i:=START_IDX TO MAX_NUM_LIGHTS BY 1 DO

			// Manual Light trigger
			// exposuretime
			IF hmi.in.recipe.useCamExpTimeForLight THEN
				hw.lights[i].out.par.exposureTime := hmi.in.recipe.cam.exposureTime;
			ELSE
				hw.lights[i].out.par.exposureTime := hmi.in.recipe.lights[i].exposureTime;
			END_IF
			// color
			IF hmi.in.recipe.useCamLedColorForLight THEN
				hw.lights[i].out.par.flashColor := hmi.in.recipe.cam.flashColor;
			ELSE
				hw.lights[i].out.par.flashColor := hmi.in.recipe.lights[i].flashColor;
			END_IF

			hmi.out.lights[i].common:=hw.lights[i].in.common;
			hmi.out.lights[i].status:=hw.lights[i].in.status;
			hw.lights[i].out.par.flashAngle:=hmi.in.recipe.lights[i].flashAngle;

			hmi.out.lights[i].plNodeNr := idx*16+UINT_TO_USINT(i-1);

			IF hmi.in.cmd.lights[i].flashTrigger AND NOT hw.lights[i].out.cmd.flashTrigger THEN
				hmi.in.cmd.lights[i].flashTrigger := FALSE;
				hw.lights[i].out.cmd.flashTrigger := TRUE;

				// Nettime
				hw.lights[i].out.par.nettime := hw.io.in.nettime + gAxis.status.powerlinkCycleTime * commonHmi.in.recipe.visionPreTriggerCycles;
			ELSIF 	hw.lights[i].out.cmd.flashTrigger AND hw.lights[i].out.par.nettime <= hw.io.in.nettime THEN
				hw.lights[i].out.cmd.flashTrigger := FALSE;
			END_IF
		END_FOR

		// -----------------------------------------------------------------------------------------------------------
		// New image ready and results
		// -----------------------------------------------------------------------------------------------------------
		// New image (hight for one scan)
		IF this.brdkViBase_imgTrigger_0.newImage THEN

			this.mappView.updateImage := NOT hmi.in.recipe.showOnlyLastImage OR this.currentTriggerNum = hmi.in.recipe.multiCaptureNum; // Trigger an update of the image on hmi
			this.DTGetTime_0(enable := TRUE);

			processResultsAction; // Process results action

			userResultProcessingAction; // User defined process results

		END_IF

		// -----------------------------------------------------------------------------------------------------------
		// Selection of specific result
		// -----------------------------------------------------------------------------------------------------------
		IF hmi.in.cmd.click THEN
			hmi.in.cmd.click := FALSE;

			//VF
			brdkStrSubStr(ADR(tmpVF),ADR(hmi.in.cmd.elemId),1,1);
			//ID
			brsstrcpy(ADR(tmpID),ADR(hmi.in.cmd.elemId)+2);

			hmi.in.cmd.intElemId := STRING_TO_USINT(tmpID);
			IF hmi.in.cmd.intElemId > MAX_NUM_RESULTS THEN
				hmi.in.cmd.intElemId := 0;
			END_IF

		END_IF

		IF hmi.in.cmd.intElemId <> this.oldIntElemID THEN
			this.oldIntElemID := hmi.in.cmd.intElemId;
			processResultsAction;
		END_IF

		// -----------------------------------------------------------------------------------------------------------
		// Auto search vision acquistion settings done (save found settings in recipe structure)
		// -----------------------------------------------------------------------------------------------------------

		// search Auto Focus done (hight for one scan)
		IF this.brdkViBase_imgTrigger_0.searchAcquisitonSettingsDone THEN
			hmi.in.cmd.autoSearch 			:= FALSE;
			hmi.in.recipe.cam.gainLevel 	:=	 hw.camera.in.status.gainLevel;
			hmi.in.recipe.cam.focus		 	:=	 hw.camera.in.status.focus;
			hmi.in.recipe.cam.exposureTime 	:=	 hw.camera.in.status.exposureTime;
			this.brdkViBase_imgTrigger_0.searchAcquisitonSettings := FALSE;
			hmi.in.cmd.trigger 				:= TRUE;
		END_IF

		// -----------------------------------------------------------------------------------------------------------
		// MappView get image to show om hmi
		// -----------------------------------------------------------------------------------------------------------

		IF DiagCpuIsSimulated() THEN
			this.mappView.imageFormat := BRDKVIIMG_IMG_TYPE_JPEG;
		ELSE
			this.mappView.imageFormat := commonHmi.in.recipe.imageFormat;
		END_IF
		this.mappView.jpegQuality := commonHmi.in.recipe.jpegQuality;
		this.mappView();

		// -----------------------------------------------------------------------------------------------------------
		// Save image to file devive F:/images
		// -----------------------------------------------------------------------------------------------------------
		CASE this.saveState OF
			0:

				IF (hmi.in.cmd.saveImage OR (this.mappView.newSvgReady AND commonHmi.in.recipe.saveAllImages))  AND gFiles.output.ready THEN
					hmi.in.cmd.saveImage := FALSE;

					// create filename with VF name and current date of the image
					brsstrcpy(ADR(this.tmpFileName),ADR(hmi.out.camera.visionFunction));
					brsstrcat(ADR(this.tmpFileName),ADR('-'));
					brdkViBase_dateTimeToString(this.DTGetTime_0.DT1,'%Y-%m-%d-%H-%M-%S',ADR(this.tmpFileName));

					brsstrcpy(ADR(this.brdkFileWrite.fileName),ADR(this.tmpFileName));

					CASE this.mappView.imageFormat OF
						BRDKVIIMG_IMG_TYPE_JPEG:
							brsstrcat(ADR(this.brdkFileWrite.fileName),ADR('.jpg'));
						BRDKVIIMG_IMG_TYPE_BMP:
							brsstrcat(ADR(this.brdkFileWrite.fileName),ADR('.bmp'));
					END_CASE

					this.brdkFileWrite.enable := TRUE;
					this.brdkFileWrite.dataLength := this.mappView.internal.getImage.destLen;
					this.brdkFileWrite.pData := this.mappView.internal.getImage.pDest;
					this.brdkFileWrite.overwrite := TRUE;
					this.brdkFileWrite.fileDevice := 'IMG';

					this.saveState := 10;
				END_IF
			10:

				IF this.brdkFileWrite.done THEN
					gFiles.input.refresh := TRUE;
					this.brdkFileWrite.enable := FALSE;
					this.saveState := 20;
				END_IF

			20:
				brsstrcpy(ADR(this.brdkFileWrite.fileName),ADR(this.tmpFileName));

				brsstrcat(ADR(this.brdkFileWrite.fileName),ADR('.svg'));
				this.brdkFileWrite.enable := TRUE;
				this.brdkFileWrite.dataLength := brsstrlen(ADR(hmi.out.svgOverlay));
				this.brdkFileWrite.pData := ADR(hmi.out.svgOverlay);
				this.brdkFileWrite.overwrite := TRUE;
				this.brdkFileWrite.fileDevice := 'IMG';

				this.saveState := 30;

			30:
				IF this.brdkFileWrite.done THEN
					gFiles.input.refresh := TRUE;
					this.brdkFileWrite.enable := FALSE;
					this.saveState := 0;
				END_IF

		END_CASE

		this.brdkFileWrite();

		// -----------------------------------------------------------------------------------------------------------
		// Save diagnostic data
		// -----------------------------------------------------------------------------------------------------------
		IF hmi.in.cmd.saveDiagnositc AND gFiles.output.ready THEN
			hmi.in.cmd.saveDiagnositc 			:= FALSE;

			// Delete old file first
			this.fileDelete.enable 					:= TRUE;
			this.fileDelete.pDevice 				:= ADR(this.visionDiagFileDevice);
			this.fileDelete.pName 					:= ADR(hmi.in.diagnosticFilename);

			// Upload diagnostic information
			this.viBaseSaveDiagData_0.MpLink 		:= this.mappView.pMappLink;
			this.viBaseSaveDiagData_0.DeviceName 	:= ADR(this.visionDiagFileDevice);
			this.viBaseSaveDiagData_0.FileName 		:= ADR(hmi.in.diagnosticFilename);
			hmi.out.camera.saveDiagStatus 			:= UINT_TO_DINT(ERR_FUB_BUSY);
		END_IF

		// file delete done or error (if file do not exsist)
		IF (this.fileDelete.enable AND this.fileDelete.status = ERR_OK) THEN
			this.fileDelete.enable 				:= FALSE;
			this.viBaseSaveDiagData_0.Execute 	:= TRUE;
		END_IF

		// Done
		IF (this.viBaseSaveDiagData_0.Done) THEN
			hmi.out.camera.saveDiagStatus		:= UINT_TO_DINT(ERR_OK);
			this.viBaseSaveDiagData_0.Execute 	:= FALSE;
		END_IF

		// Error
		IF (NOT this.viBaseSaveDiagData_0.Busy AND this.viBaseSaveDiagData_0.Error) THEN
			hmi.out.camera.saveDiagStatus		:= this.viBaseSaveDiagData_0.StatusID;
			this.viBaseSaveDiagData_0.Execute 	:= FALSE;
		END_IF

		this.viBaseSaveDiagData_0();
		this.fileDelete();

		// -----------------------------------------------------------------------------------------------------------
		// Get Vision application list from camera
		// -----------------------------------------------------------------------------------------------------------

		// trigger
		IF hmi.in.cmd.vaList.refresh THEN
			hmi.in.cmd.vaList.refresh 	:= FALSE;

			this.getVaList.Execute 		:= TRUE;
			this.getVaList.Format 		:= viBASE_FORMAT_PLAIN_TEXT;
			this.getVaList.List 		:= ADR(hmi.out.vaList.list);
			this.getVaList.ListLen 		:= SIZEOF(hmi.out.vaList.list);
			this.getVaList.MpLink 		:= this.mappView.pMappLink;
		END_IF

		// Done
		IF this.getVaList.Done THEN
			this.getVaList.Execute 		:= FALSE;
			hmi.out.vaList.length 		:= this.getVaList.NrEntries;
		END_IF

		// Error
		IF this.getVaList.Error THEN
			this.getVaList.Execute 		:= FALSE;
			hmi.out.vaList.lastError 	:= this.getVaList.StatusID;
		END_IF

		this.getVaList();

		// -----------------------------------------------------------------------------------------------------------
		// Load vision application
		// -----------------------------------------------------------------------------------------------------------

		// Trigger
		IF hmi.in.cmd.vaList.load AND brsstrlen(ADR(hmi.out.vaList.list[hmi.in.cmd.vaList.selectedIndex])) > 5 THEN
			hmi.in.cmd.vaList.load 						:= FALSE;

			this.viBaseLoadApplication_0.Execute 	:= TRUE;
			this.viBaseLoadApplication_0.MpLink		:= this.mappView.pMappLink;
			this.viBaseLoadApplication_0.Name		:= ADR(hmi.out.vaList.list[hmi.in.cmd.vaList.selectedIndex]);
			hmi.out.camera.vaLoad 					:= UINT_TO_DINT(ERR_FUB_BUSY);
		ELSE
			hmi.in.cmd.vaList.load := FALSE;
		END_IF

		// Done
		IF (this.viBaseLoadApplication_0.Done) THEN
			hmi.in.cmd.vaList.selectedIndex := 0;
			this.viBaseLoadApplication_0.Execute 	:= FALSE;
			hmi.out.camera.vaLoad 					:= UINT_TO_DINT(ERR_OK);
		END_IF

		// Error
		IF (NOT this.viBaseLoadApplication_0.Busy AND this.viBaseLoadApplication_0.Error) THEN
			this.viBaseLoadApplication_0.Execute 	:= FALSE;
			hmi.out.camera.vaLoad 					:= this.viBaseLoadApplication_0.StatusID;
		END_IF

		this.viBaseLoadApplication_0();

		// -----------------------------------------------------------------------------------------------------------
		// HMI stuff
		// -----------------------------------------------------------------------------------------------------------
		hmiAction;

		// -----------------------------------------------------------------------------------------------------------
		// Recipe handling (register recipse data structure
		// -----------------------------------------------------------------------------------------------------------
		this.mpRecipeRegVar.Enable 		:= gRecipe.out.active;
		this.mpRecipeRegVar.MpLink 		:= gRecipe.out.mpLink;
		this.mpRecipeRegVar.ConfirmSave := this.mpRecipeRegVar.SaveNotification;
		this.mpRecipeRegVar.Category 	:= ADR('Recipe');
		this.mpRecipeRegVar.PVName 		:= ADR(this.recipePVName);
		this.mpRecipeRegVar();

		// handle conversion from CR dropDown value to interger and back
		IF this.mpRecipeRegVar.UpdateNotification THEN
			hmi.in.recipe.CRTypeStr := USINT_TO_STRING(hmi.in.recipe.CR.symbolType);

			FOR i:=START_IDX TO MAX_NUM_LIGHTS BY 1 DO
				this.brdkViBase_getLightInfo[i]();
				hmi.in.cmd.lightColorStr[i] := USINT_TO_STRING(hmi.in.recipe.lights[i].flashColor );
			END_FOR

		ELSE
			hmi.in.recipe.CR.symbolType := STRING_TO_USINT(hmi.in.recipe.CRTypeStr);
			FOR i:=START_IDX TO MAX_NUM_LIGHTS BY 1 DO
				this.brdkViBase_getLightInfo[i]();
				hmi.in.recipe.lights[i].flashColor := STRING_TO_USINT(hmi.in.cmd.lightColorStr[i]);
			END_FOR
		END_IF

		// Clear ready for init (auto load) if data structures have not been registred
		IF NOT this.mpRecipeRegVar.Active THEN
			gRecipe.in.readyForInit := FALSE;
		END_IF

		userLocalPostAction; // user local action after all other

	END_FOR

	userCommonPostAction; // user common action after all other

	// -----------------------------------------------------------------------------------------------------------
	//Configure the pointers (this,hmi,hw etc.) show the correct data for that watch index
	// -----------------------------------------------------------------------------------------------------------
	watchIdx := LIMIT(START_IDX,watchIdx,MAX_NUM_CAMS);
	idx := watchIdx;
	setupPointersAction;

					END_PROGRAM

PROGRAM _EXIT

	FOR idx:= START_IDX TO MAX_NUM_CAMS BY 1 DO
		setupPointersAction;

		this.mappView(enable := FALSE);
		this.mpRecipeRegVar(Enable := FALSE);

		userExitLocalPostAction;
	END_FOR

	userExitCommonPostAction;

					END_PROGRAM
```

#### Types.typ
```iecst
(*Local data structure*)

TYPE
	local_axisTrig_typ : 	STRUCT
		nettimeLastCycle_us : DINT;
		powerlinkCycle_us : DINT;
		axisPositionNow : REAL;
		triggerPosDelta : REAL;
		triggerTimeDelta : DINT; (*In us*)
	END_STRUCT;
	local_vaList_typ : 	STRUCT
	END_STRUCT;
	local_typ : 	STRUCT
		path : STRING[100];
		lightPath : ARRAY[START_IDX..MAX_NUM_LIGHTS]OF STRING[100];
		brdkViBase_imgTrigger_0 : brdkViBase_imgTrigger;
		brdkViBase_getLightInfo : ARRAY[START_IDX..MAX_NUM_LIGHTS]OF brdkViBase_getLightInfo;
		brdkViBase_getCameraInfo_0 : brdkViBase_getCameraInfo;
		mappView : {REDUND_UNREPLICABLE} brdkViImg_mappView;
		viBaseSaveDiagData_0 : ViBaseSaveDiagData;
		fileDelete : FileDelete;
		visionDiagFileDevice : STRING[10];
		viBaseLoadApplication_0 : ViBaseLoadApplication;
		axisTrig : local_axisTrig_typ;
		brdkFileWrite : brdkFileWrite;
		dtNow : DTStructure;
		DTGetTime_0 : DTGetTime;
		tmp2D : brdkViBase_2d_typ;
		strElemId : STRING[80];
		oldIntElemID : USINT;
		elemId : STRING[80];
		tmpAngle : LREAL;
		strStyle : STRING[240];
		mpRecipeRegVar : MpRecipeRegParSync;
		recipePVName : STRING[100];
		getVaList : ViBaseListApplication;
		tmpFileName : STRING[255];
		saveState : USINT;
		ioTrigger : R_TRIG;
		user : user_local_typ;
		currentTriggerNum : UINT;
		repetitiveTriggerTON : TON;
		tmpDraw : hmi_in_recipe_draw_typ;
	END_STRUCT;
END_TYPE

(*Hardware*)

TYPE
	hw_io_in_typ : 	STRUCT
		nettime : DINT;
		commonTrigger : BOOL;
		individualTrigger : BOOL;
	END_STRUCT;
	hw_io_typ : 	STRUCT
		in : hw_io_in_typ;
	END_STRUCT;
	hw_typ : 	STRUCT
		camera : brdkViBase_cam_hw_typ;
		VF : hw_VF_typ;
		lights : ARRAY[START_IDX..MAX_NUM_LIGHTS]OF brdkViBase_light_hw_typ;
		io : hw_io_typ;
		user : user_hw_typ;
	END_STRUCT;
	hw_VF_typ : 	STRUCT
		codeReader : brdkViBase_hw_cr_10_typ;
		pixelCnt : brdkViBase_hw_pxCnt_10_typ;
		measurement : brdkViBase_hw_meas_10_typ;
		matching : brdkViBase_hw_match_10_typ;
		ocr : brdkViBase_hw_OCR_10_typ;
		blob : brdkViBase_hw_blob_10_typ;
	END_STRUCT;
END_TYPE

(*HMI*)

TYPE
	hmi_typ : 	STRUCT
		in : hmi_in_typ;
		out : hmi_out_typ;
		user : user_hmi_typ;
	END_STRUCT;
END_TYPE

(*HMI output*)

TYPE
	hmi_out_typ : 	STRUCT
		svgOverlay : STRING[10000];
		wsPort : UINT;
		lights : ARRAY[START_IDX..MAX_NUM_LIGHTS]OF hmi_out_lights_typ;
		camera : hmi_out_camera_typ;
		VF : hmi_out_vf_typ;
		tableVF : hmi_out_vf_table_typ;
		vaList : hmi_out_vaList_typ;
		usedVF : hmi_out_usedVF_typ;
	END_STRUCT;
	hmi_out_vf_typ : 	STRUCT
		processingTime : UDINT;
		numResults : USINT;
		match : brdkViBase_hmi_match_in_typ;
		measurement : brdkViBase_hw_meas_in_typ;
		codeReader : brdkViBase_hmi_cr_in_typ;
		ocr : brdkViBase_hmi_OCR_in_typ;
		pixelCnt : brdkViBase_hmi_pxCnt_in_typ;
		blob : brdkViBase_hmi_blob_in_typ;
	END_STRUCT;
	hmi_out_lights_typ : 	STRUCT
		status : brdkViBase_light_hw_status_typ;
		common : brdkViBase_hw_in_common_typ;
		simulated : BOOL;
		connectedText : STRING[20];
		connected : BOOL;
		statusText : STRING[50];
		lightType : USINT;
		plNodeNr : USINT;
		info : brdkViBase_lightInfo_typ;
		flashLightOptions : ARRAY[0..4]OF STRING[50];
	END_STRUCT;
	hmi_out_camera_typ : 	STRUCT
		simulated : BOOL;
		connectedText : STRING[20];
		connected : BOOL;
		mappVisionActive : BOOL;
		processing : BOOL;
		ready : BOOL;
		statusText : STRING[50];
		plNodeNr : USINT;
		visionFunction : STRING[20];
		processingTime : UDINT;
		opticInfo : brdkViBase_opticInfo_typ;
		common : brdkViBase_hw_in_common_typ;
		hw : brdkViBase_cam_hw_in_status_typ;
		vaLoad : DINT;
		saveDiagStatus : DINT;
		flashLightOptions : ARRAY[0..4]OF STRING[50];
	END_STRUCT;
	hmi_out_vaList_typ : 	STRUCT
		list : ARRAY[0..99]OF ViBaseFormatPlainTextType;
		length : {REDUND_UNREPLICABLE} UINT;
		lastError : DINT;
	END_STRUCT;
	hmi_out_usedVF_typ : 	STRUCT
		pixelCounter : BOOL;
		measurement : BOOL;
		matching : BOOL;
		codeReader : BOOL;
		OCR : BOOL;
		BLOB : BOOL;
	END_STRUCT;
	hmi_out_vf_table_cr_typ : 	STRUCT  (*Code reader structures*)
		BarcodeText : ARRAY[START_IDX..MAX_NUM_RESULTS]OF STRING[101];
		BarcodeType : ARRAY[START_IDX..MAX_NUM_RESULTS]OF USINT;
		PositionX : ARRAY[START_IDX..MAX_NUM_RESULTS]OF REAL;
		PositionY : ARRAY[START_IDX..MAX_NUM_RESULTS]OF REAL;
		Orientation : ARRAY[START_IDX..MAX_NUM_RESULTS]OF REAL;
		Grading : ARRAY[START_IDX..MAX_NUM_RESULTS]OF SINT;
	END_STRUCT;
	hmi_out_vf_table_blob_typ : 	STRUCT  (*Blob function structures*)
		ModelNumber : ARRAY[START_IDX..MAX_NUM_RESULTS]OF USINT;
		Clipped : ARRAY[START_IDX..MAX_NUM_RESULTS]OF BOOL;
		Area : ARRAY[START_IDX..MAX_NUM_RESULTS]OF REAL;
		PositionX : ARRAY[START_IDX..MAX_NUM_RESULTS]OF REAL;
		PositionY : ARRAY[START_IDX..MAX_NUM_RESULTS]OF REAL;
		Orientation : ARRAY[START_IDX..MAX_NUM_RESULTS]OF REAL;
		MeanGrayValue : ARRAY[START_IDX..MAX_NUM_RESULTS]OF USINT;
		Length : ARRAY[START_IDX..MAX_NUM_RESULTS]OF UDINT;
		Width : ARRAY[START_IDX..MAX_NUM_RESULTS]OF UDINT;
	END_STRUCT;
	hmi_out_vf_match_typ : 	STRUCT  (*Match function structures*)
		ModelNumber : ARRAY[START_IDX..MAX_NUM_RESULTS]OF USINT;
		Score : ARRAY[START_IDX..MAX_NUM_RESULTS]OF REAL;
		PositionX : ARRAY[START_IDX..MAX_NUM_RESULTS]OF REAL;
		PositionY : ARRAY[START_IDX..MAX_NUM_RESULTS]OF REAL;
		Orientation : ARRAY[START_IDX..MAX_NUM_RESULTS]OF REAL;
		Scale : ARRAY[START_IDX..MAX_NUM_RESULTS]OF REAL;
		RotCenterX : ARRAY[START_IDX..MAX_NUM_RESULTS]OF REAL;
		RotCenterY : ARRAY[START_IDX..MAX_NUM_RESULTS]OF REAL;
	END_STRUCT;
	hmi_out_vf_table_ocr_typ : 	STRUCT  (*OCR function structures*)
		Text : ARRAY[START_IDX..MAX_NUM_RESULTS]OF STRING[51];
		Grading : ARRAY[START_IDX..MAX_NUM_RESULTS]OF USINT;
		PositionX : ARRAY[START_IDX..MAX_NUM_RESULTS]OF REAL;
		PositionY : ARRAY[START_IDX..MAX_NUM_RESULTS]OF REAL;
		Orientation : ARRAY[START_IDX..MAX_NUM_RESULTS]OF REAL;
	END_STRUCT;
	hmi_out_vf_table_pxCnt_typ : 	STRUCT  (*OCR function structures*)
		ModelNumber : ARRAY[START_IDX..MAX_NUM_RESULTS]OF USINT;
		NumPixels : ARRAY[START_IDX..MAX_NUM_RESULTS]OF UDINT;
		MinGray : ARRAY[START_IDX..MAX_NUM_RESULTS]OF USINT;
		MaxGray : ARRAY[START_IDX..MAX_NUM_RESULTS]OF USINT;
		MeanGray : ARRAY[START_IDX..MAX_NUM_RESULTS]OF REAL;
		DeviationGray : ARRAY[START_IDX..MAX_NUM_RESULTS]OF REAL;
		MedianGray : ARRAY[START_IDX..MAX_NUM_RESULTS]OF USINT;
		ModelArea : ARRAY[START_IDX..MAX_NUM_RESULTS]OF UDINT;
		NumConnectedComponents : ARRAY[START_IDX..MAX_NUM_RESULTS]OF UINT;
		PositionX : ARRAY[START_IDX..MAX_NUM_RESULTS]OF REAL;
		PositionY : ARRAY[START_IDX..MAX_NUM_RESULTS]OF REAL;
	END_STRUCT;
	hmi_out_vf_table_meas_typ : 	STRUCT  (*MT function structures*)
		Result : ARRAY[START_IDX..MAX_NUM_RESULTS]OF DINT;
	END_STRUCT;
	hmi_out_vf_table_typ : 	STRUCT
		match : hmi_out_vf_match_typ;
		ocr : hmi_out_vf_table_ocr_typ;
		measurement : hmi_out_vf_table_meas_typ;
		pixelCnt : hmi_out_vf_table_pxCnt_typ;
		blob : hmi_out_vf_table_blob_typ;
		codeReader : hmi_out_vf_table_cr_typ;
		tableNum : ARRAY[START_IDX..MAX_NUM_RESULTS]OF USINT;
	END_STRUCT;
END_TYPE

(*HMI Input*)

TYPE
	hmi_in_typ : 	STRUCT
		cmd : hmi_in_cmd_typ;
		recipe : recipe_typ;
		cameraInfo : brdkViBase_camInfo_typ;
		diagnosticFilename : STRING[50];
		vaName : STRING[50];
		lightNum : USINT := 1;
	END_STRUCT;
	hmi_in_cmd_flashSegment_typ : 	STRUCT
		top : BOOL := TRUE;
		bottom : BOOL := TRUE;
		right : BOOL := TRUE;
		left : BOOL := TRUE;
	END_STRUCT;
	hmi_in_cmd_vaList_typ : 	STRUCT
		refresh : BOOL;
		selectedIndex : UINT;
		load : BOOL;
	END_STRUCT;
	hmi_in_cmd_typ : 	STRUCT
		lights : ARRAY[START_IDX..MAX_NUM_LIGHTS]OF brdkViBase_light_hw_out_cmd_typ;
		flashSegment : hmi_in_cmd_flashSegment_typ;
		trigger : BOOL; (*Trigger a image*)
		autoSearch : BOOL; (*Start auto Search of exposure and focus for camra*)
		resetInfo : BOOL; (*Reset optic info to the current camera*)
		saveDiagnositc : BOOL; (*Save vision diagnostic *)
		saveImage : BOOL;
		intElemId : USINT := 1;
		elemId : STRING[80];
		click : BOOL;
		y : REAL;
		x : REAL;
		vaList : hmi_in_cmd_vaList_typ;
		resultTabIndex : USINT;
		lightColorStr : ARRAY[START_IDX..MAX_NUM_LIGHTS]OF STRING[50];
	END_STRUCT;
	hmi_in_recipe_draw_typ : 	STRUCT
		intShape : INT := 0; (*0 = None, 1=  rectangle, 2 = circle, 3 = triangle*)
		radius : REAL := 60;
		width : REAL := 80;
		length : REAL := 80;
		rotation : REAL := 0;
		fillColor : STRING[80] := ' fill: green;';
		activeStrokeColor : STRING[80] := ' stroke: orange;';
		strokeColor : STRING[80] := ' stroke: green;';
		strokeWidth : INT := 5;
		strokeOpac : REAL := 1;
		fillOpac : REAL := 0.3;
	END_STRUCT;
END_TYPE

(*Recipe data structure (saved to file and included in the HMI input data structure for access from HMI)*)

TYPE
	recipe_typ : 	STRUCT
		lights : ARRAY[START_IDX..MAX_NUM_LIGHTS]OF brdkViBase_light_hw_out_par_typ;
		cam : brdkViBase_cam_recipe_typ;
		BLOB : brdkViBase_hw_blob_out_typ;
		CR : brdkViBase_hw_cr_out_typ := (symbolType:=0);
		match : brdkViBase_hw_match_out_typ;
		meassurement : brdkViBase_hw_meas_out_typ;
		OCR : brdkViBase_hw_OCR_out_typ;
		pxCnt : brdkViBase_hw_pxCnt_out_typ;
		useCamExpTimeForLight : BOOL := TRUE;
		useCamLedColorForLight : BOOL := TRUE;
		ioTriggerDelay : DINT := 100;
		enableIoTrigger : BOOL := FALSE;
		multiCaptureNum : UINT := 1;
		showOnlyLastImage : BOOL := FALSE;
		draw : hmi_in_recipe_draw_typ;
		enableAxisTrigger : BOOL := FALSE;
		repetitiveTriggerInterval : UDINT := 1000;
		repetitiveTrigger : BOOL := FALSE;
		CRTypeStr : STRING[20] := '0';
		user : user_recipe_typ;
	END_STRUCT;
	common_recipe_typ : 	STRUCT
		jpegQuality : USINT := 50;
		imageFormat : BRDKVIIMG_IMG_TYPE := BRDKVIIMG_IMG_TYPE_JPEG;
		visionPreTriggerCycles : DINT := 12;
		enableAxisTrigger : BOOL;
		saveAllImages : BOOL;
		saveSvg : BOOL;
		saveImage : BOOL;
		user : user_common_recipe_typ;
	END_STRUCT;
END_TYPE

(*Common HMI*)

TYPE
	common_hmi_in_cmd_typ : 	STRUCT
		deleteAllImage : BOOL;
		refreshVAlist : BOOL;
	END_STRUCT;
	common_hmi_in_typ : 	STRUCT
		recipe : common_recipe_typ;
		cmd : common_hmi_in_cmd_typ;
		dataFilePostName : STRING[255];
	END_STRUCT;
	common_hmi_out_typ : 	STRUCT
		tmp : USINT;
	END_STRUCT;
	common_hmi_typ : 	STRUCT
		out : common_hmi_out_typ;
		in : common_hmi_in_typ;
		user : user_commonHmi_typ;
	END_STRUCT;
END_TYPE
```

#### Variables.var
```iecst
(*Constants*)
VAR CONSTANT
	START_IDX : USINT := 1; (*Start index of arrays *)
	MAX_NUM_RESULTS_M1 : USINT := MAX_NUM_RESULTS-1; (*Max number of results -1 *)
	MAX_NUM_RESULTS : USINT := 10; (*Max number of results*)
	MAX_NUM_CAMS : USINT := 6; (*Number of cameras*)
	MAX_NUM_LIGHTS : USINT := 9; (*Number of lights*)
END_VAR
(*Array instances*)
VAR
	hwInstance : ARRAY[START_IDX..MAX_NUM_CAMS] OF hw_typ; (*An array of hardware data structures for each camera*)
	hmiInstance : ARRAY[START_IDX..MAX_NUM_CAMS] OF hmi_typ; (*An array of HMI data structures for each camera*)
	localInstance : ARRAY[START_IDX..MAX_NUM_CAMS] OF local_typ; (*An array of local data structures for each camera*)
	commonHmi : common_hmi_typ; (*Common hmi variables that apply to all cameras*)
END_VAR
(*Pointers to array instances*)
VAR
	hw : REFERENCE TO hw_typ; (*Pointer to a hardware data structure*)
	hmi : REFERENCE TO hmi_typ; (*Pointer to a HMI data structure*)
	this : REFERENCE TO local_typ; (*Pointer to a Local data structure*)
	watchIdx : USINT; (*Used to indicate what array instance the points should point to (set at the end of the program)*)
	idx : USINT; (*Current Array index (e.g. camrea)*)
END_VAR
(*Variables used for loops*)
VAR
	i : USINT;
	u : USINT;
	k : USINT;
	p : USINT;
	j : USINT;
END_VAR
(*Temporary variables*)
VAR
	debug : BOOL;
	tmpStr : STRING[100];
	tmpVF : STRING[80];
	tmpID : STRING[80];
	pOffset : REFERENCE TO brdkviBase_hw_vf_out_offset_typ;
	id : UDINT;
END_VAR
```

#### hmiAction.st - HMI related
```iecst
ACTION hmiAction:

	// Work around untill units in compund widgets are fixed

	pOffset ACCESS ADR(hw.VF.blob.out.common.offsetROI);
	pOffset.orientation := pOffset.orientation *100;
	pOffset.rotCenterX := pOffset.rotCenterX *100;
	pOffset.rotCenterY := pOffset.rotCenterY *100;
	pOffset.x := pOffset.x *100;
	pOffset.y := pOffset.y *100;

	pOffset ACCESS ADR(hw.VF.codeReader.out.common.offsetROI);
	pOffset.orientation := pOffset.orientation *100;
	pOffset.rotCenterX := pOffset.rotCenterX *100;
	pOffset.rotCenterY := pOffset.rotCenterY *100;
	pOffset.x := pOffset.x *100;
	pOffset.y := pOffset.y *100;

	pOffset ACCESS ADR(hw.VF.matching.out.common.offsetROI);
	pOffset.orientation := pOffset.orientation *100;
	pOffset.rotCenterX := pOffset.rotCenterX *100;
	pOffset.rotCenterY := pOffset.rotCenterY *100;
	pOffset.x := pOffset.x *100;
	pOffset.y := pOffset.y *100;

	pOffset ACCESS ADR(hw.VF.measurement.out.common.offsetROI);
	pOffset.orientation := pOffset.orientation *100;
	pOffset.rotCenterX := pOffset.rotCenterX *100;
	pOffset.rotCenterY := pOffset.rotCenterY *100;
	pOffset.x := pOffset.x *100;
	pOffset.y := pOffset.y *100;

	pOffset ACCESS ADR(hw.VF.ocr.out.common.offsetROI);
	pOffset.orientation := pOffset.orientation *100;
	pOffset.rotCenterX := pOffset.rotCenterX *100;
	pOffset.rotCenterY := pOffset.rotCenterY *100;
	pOffset.x := pOffset.x *100;
	pOffset.y := pOffset.y *100;

	pOffset ACCESS ADR(hw.VF.pixelCnt.out.common.offsetROI);
	pOffset.orientation := pOffset.orientation *100;
	pOffset.rotCenterX := pOffset.rotCenterX *100;
	pOffset.rotCenterY := pOffset.rotCenterY *100;
	pOffset.x := pOffset.x *100;
	pOffset.y := pOffset.y *100;

	// Work around done

	IF DiagCpuIsSimulated() OR (NOT hw.camera.in.common.moduleOk AND this.brdkViBase_imgTrigger_0.simulate.alwaysSimulateNonePresentCamera) THEN
		hmi.out.camera.connected :=  TRUE;
		hmi.out.camera.simulated := TRUE;
	ELSE

		hmi.out.camera.simulated := FALSE;
		IF hw.camera.in.common.moduleOk THEN
			hmi.out.camera.connected :=  TRUE;
		ELSE
			hmi.out.camera.connected :=  FALSE;
		END_IF
	END_IF
	hmi.out.camera.processing := hw.camera.in.status.imageProcessingActive;
	hmi.out.camera.ready := this.brdkViBase_imgTrigger_0.ready AND NOT hmi.in.recipe.repetitiveTrigger;

	brsmemcpy(ADR(hmi.out.camera.hw),ADR(hw.camera.in.status),SIZEOF(hmi.out.camera.hw));
	brsmemcpy(ADR(hmi.out.camera.common),ADR(hw.camera.in.common),SIZEOF(hmi.out.camera.common));

	IF brsmemcmp(ADR(hmi.in.recipe.draw),ADR(this.tmpDraw),SIZEOF(this.tmpDraw)) <> 0 THEN
		processResultsAction;
		this.tmpDraw := hmi.in.recipe.draw;
	END_IF

	IF this.mpRecipeRegVar.UpdateNotification THEN

		hmi.in.cmd.flashSegment.top 	:= hmi.in.recipe.cam.flashSegment.0;
		hmi.in.cmd.flashSegment.bottom 	:= hmi.in.recipe.cam.flashSegment.1;
		hmi.in.cmd.flashSegment.left 	:= hmi.in.recipe.cam.flashSegment.2;
		hmi.in.cmd.flashSegment.right 	:= hmi.in.recipe.cam.flashSegment.3;

	ELSE
		hmi.in.recipe.cam.flashSegment.0 := hmi.in.cmd.flashSegment.top;
		hmi.in.recipe.cam.flashSegment.1 := hmi.in.cmd.flashSegment.bottom;
		hmi.in.recipe.cam.flashSegment.2 := hmi.in.cmd.flashSegment.left;
		hmi.in.recipe.cam.flashSegment.3 := hmi.in.cmd.flashSegment.right;
	END_IF

	IF hmi.in.cmd.intElemId > 0 THEN

		IF hmi.in.cmd.intElemId <= hw.VF.blob.in.common.numResults THEN
			brdkViBase_blob_hw2hmi(hw.VF.blob.in.results[hmi.in.cmd.intElemId-1],hmi.out.VF.blob);
		ELSE
			brsmemset(ADR(hmi.out.VF.blob),0,SIZEOF(hmi.out.VF.blob));
		END_IF

		IF hmi.in.cmd.intElemId <= hw.VF.codeReader.in.common.numResults THEN
			brdkViBase_cr_hw2hmi(hw.VF.codeReader.in.results[hmi.in.cmd.intElemId-1],hmi.out.VF.codeReader);
		ELSE
			brsmemset(ADR(hmi.out.VF.codeReader),0,SIZEOF(hmi.out.VF.codeReader));
		END_IF

		IF hmi.in.cmd.intElemId <= hw.VF.matching.in.common.numResults THEN
			brdkViBase_match_hw2hmi(hw.VF.matching.in.results[hmi.in.cmd.intElemId-1],hmi.out.VF.match);
		ELSE
			brsmemset(ADR(hmi.out.VF.match),0,SIZEOF(hmi.out.VF.match));
		END_IF

		IF hmi.in.cmd.intElemId <= hw.VF.measurement.in.common.numResults THEN
			brdkViBase_meas_hw2hmi(hw.VF.measurement.in.results[hmi.in.cmd.intElemId-1],hmi.out.VF.measurement);
		ELSE
			brsmemset(ADR(hmi.out.VF.measurement),0,SIZEOF(hmi.out.VF.measurement));
		END_IF

		IF hmi.in.cmd.intElemId <= hw.VF.ocr.in.common.numResults THEN
			brdkViBase_ocr_hw2hmi(hw.VF.ocr.in.results[hmi.in.cmd.intElemId-1],hmi.out.VF.ocr);
		ELSE
			brsmemset(ADR(hmi.out.VF.ocr),0,SIZEOF(hmi.out.VF.ocr));
		END_IF

		IF hmi.in.cmd.intElemId <= hw.VF.pixelCnt.in.common.numResults THEN
			brdkViBase_pxCnt_hw2hmi(hw.VF.pixelCnt.in.results[hmi.in.cmd.intElemId-1],hmi.out.VF.pixelCnt);
		ELSE
			brsmemset(ADR(hmi.out.VF.pixelCnt),0,SIZEOF(hmi.out.VF.pixelCnt));
		END_IF
	ELSE
		// clear if 0
		brsmemset(ADR(hmi.out.VF.pixelCnt),0,SIZEOF(hmi.out.VF.pixelCnt));
		brsmemset(ADR(hmi.out.VF.ocr),0,SIZEOF(hmi.out.VF.ocr));
		brsmemset(ADR(hmi.out.VF.measurement),0,SIZEOF(hmi.out.VF.measurement));
		brsmemset(ADR(hmi.out.VF.match),0,SIZEOF(hmi.out.VF.match));
		brsmemset(ADR(hmi.out.VF.blob),0,SIZEOF(hmi.out.VF.blob));
		brsmemset(ADR(hmi.out.VF.codeReader),0,SIZEOF(hmi.out.VF.codeReader));
	END_IF

END_ACTION
```

#### processResultsAction.st - Process the vision results and draw overlay
```iecst
ACTION processResultsAction:

	this.tmpAngle:= -(hmi.in.recipe.draw.rotation);

	// DRAW CIRCLES ON RESULTS
	hmi.out.svgOverlay := '';
	brsmemset(ADR(hmi.out.tableVF),0,SIZEOF(hmi.out.tableVF));

	//BLOB
	IF hw.VF.blob.in.common.numResults > 0 THEN
		FOR i:= 1 TO hw.VF.blob.in.common.numResults BY 1 DO

			//----------------------------------
			//          table results
			hmi.out.tableVF.blob.ModelNumber[i] := hw.VF.blob.in.results[i-1].modelNumber;
			hmi.out.tableVF.blob.Clipped[i] := hw.VF.blob.in.results[i-1].clipped;
			hmi.out.tableVF.blob.Area[i] := hw.VF.blob.in.results[i-1].area;
			hmi.out.tableVF.blob.PositionX[i] := DINT_TO_REAL(hw.VF.blob.in.results[i-1].positionX) /100.0;
			hmi.out.tableVF.blob.PositionY[i] :=  DINT_TO_REAL(hw.VF.blob.in.results[i-1].positionY) /100.0;
			hmi.out.tableVF.blob.Orientation[i] :=  DINT_TO_REAL(hw.VF.blob.in.results[i-1].orientation) /100.0;
			hmi.out.tableVF.blob.MeanGrayValue[i] := hw.VF.blob.in.results[i-1].meanGreyValue;
			hmi.out.tableVF.blob.Length[i] := hw.VF.blob.in.results[i-1].length;
			hmi.out.tableVF.blob.Width[i] := hw.VF.blob.in.results[i-1].width;

			//------------------------------------
			//			Overlay darwing
			this.tmp2D.x := DINT_TO_REAL(hw.VF.blob.in.results[i-1].positionX) / 100.0;
			this.tmp2D.y := DINT_TO_REAL(hw.VF.blob.in.results[i-1].positionY) / 100.0;
			this.tmpAngle:= -(hmi.out.tableVF.blob.PositionY[i]);
			// Style string generation
			// e.g.:'id="13" style="fill:blue;stroke:blue;stroke-width:5;fill-opacity:0.3;stroke-opacity:1"'
			this.strStyle := 'id="1';

			// Draw selested shape with specified parameters on the overlay
			styleStringGeneration;
		END_FOR;
	END_IF

	//CODE READER

	IF hw.VF.codeReader.in.common.numResults > 0 THEN
		FOR i:= 1 TO hw.VF.codeReader.in.common.numResults BY 1 DO

			//----------------------------------
			//          table results
			//Conversion of individual USINT values into strings for Code Reader
			brsmemcpy(ADR(hmi.out.tableVF.codeReader.BarcodeText[i]),ADR(hw.VF.codeReader.in.results[i-1].data),SIZEOF(hw.VF.codeReader.in.results[i-1].data));
			hmi.out.tableVF.codeReader.BarcodeType[i] 		:= hw.VF.codeReader.in.results[i-1].symbolType;
			hmi.out.tableVF.codeReader.Grading[i] 		:= hw.VF.codeReader.in.results[i-1].gradingValue;
			hmi.out.tableVF.codeReader.PositionX[i] 	:=  DINT_TO_REAL(hw.VF.codeReader.in.results[i-1].positionX) /100.0;
			hmi.out.tableVF.codeReader.PositionY[i] 	:=  DINT_TO_REAL(hw.VF.codeReader.in.results[i-1].positionY) /100.0;
			hmi.out.tableVF.codeReader.Orientation[i] 	:=  DINT_TO_REAL(hw.VF.codeReader.in.results[i-1].orientation) /100.0;

			//------------------------------------
			//			Overlay darwing

			this.tmp2D.x := DINT_TO_REAL(hw.VF.codeReader.in.results[i-1].positionX) / 100.0;
			this.tmp2D.y := DINT_TO_REAL(hw.VF.codeReader.in.results[i-1].positionY) / 100.0;
			this.tmpAngle:= -REAL_TO_LREAL(hmi.out.tableVF.codeReader.Orientation[i]);

			// Style string generation
			// e.g.:'id="13" style="fill:blue;stroke:blue;stroke-width:5;fill-opacity:0.3;stroke-opacity:1"'
			this.strStyle := 'id="2';

			styleStringGeneration;
		END_FOR;
	END_IF;

	//MATCHING

	IF hw.VF.matching.in.common.numResults > 0 THEN
		FOR i:= 1 TO hw.VF.matching.in.common.numResults BY 1 DO

			//----------------------------------
			//          table results
			hmi.out.tableVF.match.ModelNumber[i] := hw.VF.matching.in.results[i-1].modelNumber;
			hmi.out.tableVF.match.Score[i] :=  DINT_TO_REAL(hw.VF.matching.in.results[i-1].score);
			hmi.out.tableVF.match.PositionX[i] :=  DINT_TO_REAL(hw.VF.matching.in.results[i-1].positionX) /100.0;
			hmi.out.tableVF.match.PositionY[i] :=  DINT_TO_REAL(hw.VF.matching.in.results[i-1].positionY) /100.0;
			hmi.out.tableVF.match.Orientation[i] :=  DINT_TO_REAL(hw.VF.matching.in.results[i-1].orientation) /100.0;
			hmi.out.tableVF.match.Scale[i] :=  DINT_TO_REAL(hw.VF.matching.in.results[i-1].scale);

			//------------------------------------
			//			Overlay darwing

			this.tmp2D.x := DINT_TO_REAL(hw.VF.matching.in.results[i-1].positionX) / 100.0;
			this.tmp2D.y := DINT_TO_REAL(hw.VF.matching.in.results[i-1].positionY) / 100.0;
			this.tmpAngle:= -REAL_TO_LREAL(hmi.out.tableVF.match.Orientation[i]+hmi.in.recipe.draw.rotation);
			// Style string generation
			// e.g.:'id="13" style="fill:blue;stroke:blue;stroke-width:5;fill-opacity:0.3;stroke-opacity:1"'
			this.strStyle := 'id="3';

			// DRAW SELECTED SHAPE WITH SPECIFIED PARAMETERS ON THE OVERLAY
			styleStringGeneration;

		END_FOR;
	END_IF;

	//MEASUREMENT

	IF hw.VF.measurement.in.common.numResults > 0 THEN
		FOR i:=1 TO hw.VF.measurement.in.common.numResults DO
			hmi.out.tableVF.measurement.Result[i] := hw.VF.measurement.in.results[i-1].result;
		END_FOR;
	END_IF;

	//OCR

	IF hwInstance[5].VF.ocr.in.common.numResults > 0 THEN
		FOR i:= 1 TO hw.VF.ocr.in.common.numResults BY 1 DO
			//----------------------------------
			//          table results
			hmi.out.tableVF.ocr.Grading[i] := hw.VF.ocr.in.results[i-1].gradingValue;
			hmi.out.tableVF.ocr.PositionX[i] :=  DINT_TO_REAL(hw.VF.ocr.in.results[i-1].positionX) /100.0;
			hmi.out.tableVF.ocr.PositionY[i] :=  DINT_TO_REAL(hw.VF.ocr.in.results[i-1].positionY) /100.0;
			hmi.out.tableVF.ocr.Orientation[i] :=  DINT_TO_REAL(hw.VF.ocr.in.results[i-1].orientation) /100.0;
			//Conversion of individual USINT values into strings for OCR
			brsmemcpy(ADR(hmi.out.tableVF.ocr.Text[i]),ADR(hw.VF.ocr.in.results[i-1].data),SIZEOF(hw.VF.ocr.in.results[i-1].data));

			//------------------------------------
			//			Overlay darwing

			this.tmp2D.x := DINT_TO_REAL(hw.VF.ocr.in.results[i-1].positionX) / 100.0;
			this.tmp2D.y := DINT_TO_REAL(hw.VF.ocr.in.results[i-1].positionY) / 100.0;
			this.tmpAngle:= -REAL_TO_LREAL(hmi.out.tableVF.ocr.PositionY[i]);
			// Style string generation
			// e.g.:'id="13" style="fill:blue;stroke:blue;stroke-width:5;fill-opacity:0.3;stroke-opacity:1"'

			this.strStyle := 'id="5';

			// DRAW SELECTED SHAPE WITH SPECIFIED PARAMETERS ON THE OVERLAY
			styleStringGeneration;

		END_FOR;
	END_IF;

	//PIXEL COUNT

	IF hwInstance[6].VF.pixelCnt.in.common.numResults > 0 THEN
		FOR i:= 1 TO hw.VF.pixelCnt.in.common.numResults BY 1 DO
			//----------------------------------
			//          table results
			hmi.out.tableVF.pixelCnt.ModelNumber[i] := hw.VF.pixelCnt.in.results[i-1].modelNumber;
			hmi.out.tableVF.pixelCnt.ModelArea[i] := hw.VF.pixelCnt.in.results[i-1].modelArea;
			hmi.out.tableVF.pixelCnt.NumPixels[i] := hw.VF.pixelCnt.in.results[i-1].numPixels;
			hmi.out.tableVF.pixelCnt.MinGray[i] := hw.VF.pixelCnt.in.results[i-1].minGray;
			hmi.out.tableVF.pixelCnt.MaxGray[i] := hw.VF.pixelCnt.in.results[i-1].maxGray;
			hmi.out.tableVF.pixelCnt.DeviationGray[i] :=  DINT_TO_REAL(hw.VF.pixelCnt.in.results[i-1].deviationGray) /100.0;
			hmi.out.tableVF.pixelCnt.MeanGray[i] :=  DINT_TO_REAL(hw.VF.pixelCnt.in.results[i-1].meanGray) /100.0;
			hmi.out.tableVF.pixelCnt.NumConnectedComponents[i] := hw.VF.pixelCnt.in.results[i-1].numConnectedComponents;
			hmi.out.tableVF.pixelCnt.PositionX[i] := DINT_TO_REAL(hw.VF.pixelCnt.in.results[i-1].positionX) /100.0;
			hmi.out.tableVF.pixelCnt.PositionY[i] := DINT_TO_REAL(hw.VF.pixelCnt.in.results[i-1].positionY) /100.0;

			//------------------------------------
			//			Overlay darwing

			this.tmp2D.x := DINT_TO_REAL(hw.VF.pixelCnt.in.results[i-1].positionX) / 100.0;
			this.tmp2D.y := DINT_TO_REAL(hw.VF.pixelCnt.in.results[i-1].positionY) / 100.0;
			this.tmpAngle := -REAL_TO_LREAL(hmi.in.recipe.draw.rotation);

			// Style string generation
			// e.g.:'id="13" style="fill:blue;stroke:blue;stroke-width:5;fill-opacity:0.3;stroke-opacity:1"'

			this.strStyle := 'id="6';

			styleStringGeneration;

		END_FOR;
	END_IF;

		END_ACTION
```

#### styleStringGeneration.st - Generate style string for vision result
```iecst
ACTION styleStringGeneration:

	IF hmi.in.recipe.draw.intShape > 0 THEN
		this.strElemId := UINT_TO_STRING(i);
		brsstrcat(ADR(this.strStyle),ADR(this.strElemId));					// string for element id attribute (value)
		brsstrcat(ADR(this.strStyle),ADR('" style="'));						// string for beginning of the style paramateres (text)
		brsstrcat(ADR(this.strStyle),ADR(hmi.in.recipe.draw.fillColor));		// string for fill color attribute (text + value)

		IF i = hmi.in.cmd.intElemId THEN
			brsstrcat(ADR(this.strStyle),ADR(hmi.in.recipe.draw.activeStrokeColor));
		ELSE
			brsstrcat(ADR(this.strStyle),ADR(hmi.in.recipe.draw.strokeColor));	// string for stroke color attribute (text + value)
		END_IF;

		brsstrcat(ADR(this.strStyle),ADR('stroke-width: ')); 				// string for stroke width attribute (text)
		tmpStr := INT_TO_STRING(hmi.in.recipe.draw.strokeWidth);
		brsstrcat(ADR(this.strStyle),ADR(tmpStr));	// string for stroke width attribute (value)
		brsstrcat(ADR(this.strStyle),ADR('; fill-opacity: ')); 				// string for fill opacity attribute (text)
		tmpStr := REAL_TO_STRING(hmi.in.recipe.draw.fillOpac);
		brsstrcat(ADR(this.strStyle),ADR(tmpStr)); 		// string for fill opacity attribute (value)
		brsstrcat(ADR(this.strStyle),ADR('; stroke-opacity: ')); 				// string for stroke opacity attribute (text)
		tmpStr := REAL_TO_STRING(hmi.in.recipe.draw.strokeOpac);
		brsstrcat(ADR(this.strStyle),ADR(tmpStr)); 	// string for stroke opacity attribute (value)
		brsstrcat(ADR(this.strStyle),ADR('"'));
	END_IF

	CASE hmi.in.recipe.draw.intShape OF
		0: // None

		1: // Rectangle
			brdkViGeom_drawSvgRectFromCP(this.tmp2D,hmi.in.recipe.draw.length,hmi.in.recipe.draw.width,this.tmpAngle,ADR(hmi.out.svgOverlay),ADR(this.strStyle));
		2: // Circle
			brdkViGeom_drawSvgCircle(this.tmp2D,hmi.in.recipe.draw.radius,ADR(hmi.out.svgOverlay),ADR(this.strStyle));
		3: // Triangle
			brdkViGeom_drawSvgTriFromCP(this.tmp2D,hmi.in.recipe.draw.length,hmi.in.recipe.draw.width,this.tmpAngle,ADR(hmi.out.svgOverlay),ADR(this.strStyle));
	END_CASE;

END_ACTION
```

#### user.typ
```iecst
TYPE
	user_local_typ : 	STRUCT
		tmp : USINT;
	END_STRUCT;
END_TYPE

(*hardware*)

TYPE
	user_hw_in_typ : 	STRUCT
		tmp : USINT;
	END_STRUCT;
	user_hw_out_typ : 	STRUCT
		tmp : USINT;
	END_STRUCT;
END_TYPE

(*HMI*)

TYPE
	user_hw_typ : 	STRUCT
		in : user_hw_in_typ;
		out : user_hw_out_typ;
	END_STRUCT;
END_TYPE

(*Common HMI*)

TYPE
	user_commonHmi_typ : 	STRUCT
		in : user_commonHmi_in_typ;
		out : user_commonHmi_out_typ;
	END_STRUCT;
	user_commonHmi_out_typ : 	STRUCT
		tmp : USINT;
	END_STRUCT;
	user_commonHmi_in_typ : 	STRUCT
		tmp : USINT;
	END_STRUCT;
END_TYPE

(*HMI*)

TYPE
	user_hmi_typ : 	STRUCT
		in : user_hmi_in_typ;
		out : user_hmi_out_typ;
	END_STRUCT;
	user_hmi_out_typ : 	STRUCT
		tmp : USINT;
	END_STRUCT;
	user_hmi_in_typ : 	STRUCT
		tmp : USINT;
	END_STRUCT;
END_TYPE

(*Recipe*)

TYPE
	user_common_recipe_typ : 	STRUCT
		tmp : USINT;
	END_STRUCT;
	user_recipe_typ : 	STRUCT
		tmp : USINT;
	END_STRUCT;
END_TYPE
```

#### userActions.st
```iecst
// INIT
// Common action  (hwInstance[], hmiInstance[] and localInstance[] as the pointers always will point to the last index
ACTION userInitCommonPreAction:

END_ACTION

// Local run for each idx action (use hw, this and hmi as they point to the current array index)
ACTION userInitLocalPostAction:

END_ACTION

// EXECUTE
// Common action brefore all other (hwInstance[], hmiInstance[] and localInstance[] as the pointers always will point to the last index
ACTION userCommonPreAction:

END_ACTION

// Common action after all other (hwInstance[], hmiInstance[] and localInstance[] as the pointers always will point to the last index
ACTION userCommonPostAction:

END_ACTION

// Local run for each idx action before all other (use hw, this and hmi as they point to the current array index)
ACTION userLocalPreAction:

END_ACTION

// Local run for each idx action after all other (use hw, this and hmi as they point to the current array index)
ACTION userLocalPostAction:

END_ACTION

// Local action that is called after the standard vision result processing is done.
ACTION userResultProcessingAction:

END_ACTION

// EXIT
// Common action (hwInstance[], hmiInstance[] and localInstance[] as the pointers always will point to the last index
ACTION userExitCommonPostAction:

END_ACTION

// Local run for each idx action (use hw, this and hmi as they point to the current array index)
ACTION userExitLocalPostAction:

END_ACTION
```

### VisionTypes.typ - not listed in the package file held
```iecst
(*-----------------------------------------------------------------------------------------------------------------------------------------*)
(*General vision structures*)

TYPE
	typVisionMain : 	STRUCT
		CMD : typVisionCommand;
		CFG : typVisionConfig;
		DAT : typVisionData;
		FCT : typVisionFunction;
		DIA : typVisionDiag;
		OPT : typVisionOptics;
		HW : typVisionHW;
	END_STRUCT;
	typVisionCommand : 	STRUCT
		ImageTrigger : BOOL;
		ImageTriggerReset : BOOL;
		AutoSetupStartStop : BOOL;
		VaSwitchApplication : BOOL;
		SaveDiagData : BOOL;
		ReadCameraInfo : BOOL;
	END_STRUCT;
	typVisionConfig : 	STRUCT
		VisionFunction : enumVisionFunction;
		PowerlinkNode : USINT;
		DataStructure : UDINT;
		ComponentLink : ViComponentType;
		ResolutionWidth_X : UINT; (*Nr of sensor pixels in x direction (width). Is always bigger than height*)
		ResolutionHeight_Y : UINT; (*Nr of sensor pixels in y direction (height). Is always smaller than width*)
	END_STRUCT;
	typVisionFunction : 	STRUCT
		ApplicationName : STRING[40];
		Status : DINT;
	END_STRUCT;
	typVisionDiag : 	STRUCT
		DiagName : STRING[80] := 'diag.tgz';
		Status : DINT;
	END_STRUCT;
	typVisionData : 	STRUCT
		Enable : BOOL := FALSE;
		MaxItemCnt : USINT := 10;
		NettimeDelay : DINT;
		Timeout : UINT := 5000;
		Gain : USINT;
		Focus : UINT;
		Exposure : UDINT;
		FlashColor : USINT := 1;
		FlashSegment : USINT := 15;
		LedColor : USINT;
		IRFilter : BOOL;
		OffsetROIX : DINT;
		OffsetROIY : DINT;
		OffsetROIRotationCenterX : DINT;
		OffsetROIRotationCenterY : DINT;
		OffsetROIOrientation : INT;
		ChromaticLock : BOOL;
		Alignment : USINT;
		AutoSetupGain : USINT;
		AutoSetupFocus : UINT;
		AutoSetupExposure : UDINT;
		AcquisitionAcceptedCnt : USINT;
		AcquisitionCompletedCnt : USINT;
		AcquisitionFailedCnt : USINT;
		LightWarningCnt : USINT;
		ImageProcessingError : UINT;
		ImageProcessingActive : BOOL;
		ImageNettime : DINT;
		ProcessingTimeCamera : UINT;
		ProcessingTimeFunction : UINT;
		ResultCnt : USINT;
		CockpitIsActive : BOOL;
		Status : UDINT;
		StatusText : STRING[30];
		Active : BOOL;
	END_STRUCT;
	typVisionOptics : 	STRUCT
		OrderNr : STRING[40];
		Binning : BOOL;
		ResolutionX : INT;
		ResolutionY : INT;
		Lens : USINT;
		Sensor : USINT;
		ValidDistance : BOOL;
		Distance_mm : LREAL;
		DistanceLens_mm : LREAL;
		HyperFocalDistance_mm : LREAL;
		PixelSize_um : LREAL;
		PixelSizeBinning_um : LREAL;
		FocalLength_mm : LREAL;
		MinObjectDist_mm : LREAL;
		MaxObjectDist_mm : LREAL;
		Aperture : LREAL;
		CircleOfConfusion_mm : LREAL;
		DepthOfFieldNearPos_mm : LREAL;
		DepthOfFieldFarPos_mm : LREAL;
		DepthOfField_mm : LREAL;
		FieldOfView_X_mm : LREAL;
		FieldOfView_Y_mm : LREAL;
		Resolution_mmPerPx : LREAL;
	END_STRUCT;
	typVisionHW : 	STRUCT
		Connected : BOOL;
		Ready : BOOL;
		DigitalInput01 : BOOL;
		DigitalOutput01 : BOOL;
		DigitalOutputStatus01 : BOOL;
		DigitalOutput02 : BOOL;
		DigitalOutputStatus02 : BOOL;
		SerialNumber : UDINT;
		ID : UDINT;
		Variant : UDINT;
		Firmware : UDINT;
		Undervoltage : BOOL;
		Temperature : SINT;
	END_STRUCT;
	enumVisionFunction :
		(
		enumFunctionNone,
		enumBlob,
		enumCoderReader,
		enumMatch,
		enumMeasurement,
		enumOCR,
		enumPixelCounter
		);
END_TYPE

(*-----------------------------------------------------------------------------------------------------------------------------------------*)
(*General Light structures*)

TYPE
	typLightMain : 	STRUCT
		CMD : typLightCommand;
		CFG : typLightConfig;
		DAT : typLightData;
		HW : typLightHW;
	END_STRUCT;
	typLightCommand : 	STRUCT
		FlashTrigger : BOOL;
		FlashTriggerReset : BOOL;
	END_STRUCT;
	typLightConfig : 	STRUCT
		LightType : enumLightType;
		PowerlinkNode : USINT;
	END_STRUCT;
	typLightData : 	STRUCT
		Enable : USINT := 1;
		FlashColor : USINT := 1;
		FlashSegment : UINT := 15;
		Exposure : UDINT := 200;
		SetAngle : UINT;
		Timeout : UINT := 5000;
		NettimeDelay : DINT;
		FlashAcceptedCnt : USINT;
		FlashCompletedCnt : USINT;
		FlashFailedCnt : USINT;
		Status : UDINT;
	END_STRUCT;
	typLightHW : 	STRUCT
		Connected : BOOL;
		Ready : BOOL;
		SerialNumber : UDINT;
		ID : UDINT;
		Variant : UDINT;
		Firmware : UDINT;
		TemperatureLED : SINT;
		TemperatureControllerBoard : SINT;
		WarningCnt : USINT;
	END_STRUCT;
	enumLightType :
		(
		enumLightNone,
		enumBacklight,
		enumLightbar
		);
END_TYPE

(*-----------------------------------------------------------------------------------------------------------------------------------------*)
(*General nettime structures*)

TYPE
	typVisionNettime : 	STRUCT
		CMD : typNettimeCommand;
		CFG : typNettimeConfig;
		DAT : typNettimeData;
	END_STRUCT;
	typNettimeCommand : 	STRUCT
		Activate : BOOL;
	END_STRUCT;
	typNettimeConfig : 	STRUCT
		AxisPeriod : LREAL; (*Units when period repeats*)
		AxisPositionTrigger : LREAL; (*Position in the period where trigger is fired*)
		AxisPositionDelay_Cycles : LREAL; (*Delay in PLK cycles for the read position from drive*)
		VisionPreTrigger_Cycles : DINT; (*Number of powerlink cycles the trigger has to be send ahead*)
	END_STRUCT;
	typNettimeData : 	STRUCT
		NettimeNext_us : DINT; (*Calculated nettime for next trigger*)
		NettimeDelta_us : DINT; (*Difference between current nettime and calculated nettime for the camera trigger*)
		AxisPosition : LREAL; (*Current axis position*)
		AxisVelocity : LREAL; (*Current axis position*)
		AxisInVelocity : BOOL; (*Indicates that the axis is moving at speed*)
		Overflow : DINT; (*Counts up when a trigger could not be set on time*)
	END_STRUCT;
END_TYPE

(*-----------------------------------------------------------------------------------------------------------------------------------------*)
(*Color detection structures*)

TYPE
	typVisionColor : 	STRUCT
		CMD : typVisionColorCommand;
		CFG : typVisionColorConfig;
		DAT : typVisionColorData;
	END_STRUCT;
	typVisionColorCommand : 	STRUCT
		Evaluate : BOOL; (*Evaluate new product and try to determine the color*)
		Teach : BOOL; (*Teach a new product and store color information*)
		ResetError : BOOL; (*Reset error state*)
	END_STRUCT;
	typVisionColorConfig : 	STRUCT
		FlashColor1 : USINT := 1; (*First flash color (red)*)
		FlashColor2 : USINT := 2; (*Second flash color (green)*)
		FlashColor3 : USINT := 3; (*Third flash color (blue)*)
		FlashColor4 : USINT := 4; (*Fourth flash color (lime)*)
		ProductName : ARRAY[1..MAX_NUM_PRODUCTS]OF STRING[80]; (*Name of the product*)
		GrayValue1 : ARRAY[1..MAX_NUM_PRODUCTS]OF UINT; (*Mean gray value for first flash color*)
		GrayValue2 : ARRAY[1..MAX_NUM_PRODUCTS]OF UINT; (*Mean gray value for second flash color*)
		GrayValue3 : ARRAY[1..MAX_NUM_PRODUCTS]OF UINT; (*Mean gray value for third flash color*)
		GrayValue4 : ARRAY[1..MAX_NUM_PRODUCTS]OF UINT; (*Mean gray value for fourth flash color*)
		TeachingIndex : UINT(1..1000)  := 1; (*Index that is currently taught*)
		MaxError : UINT := 100; (*Maximum error for all gray values*)
		MinDifference : UINT := 10; (*Minimum distance to next best value*)
	END_STRUCT;
	typVisionColorData : 	STRUCT
		GrayValue1 : UINT; (*Current mean gray value for first flash color*)
		GrayValue2 : UINT; (*Current mean gray value for second flash color*)
		GrayValue3 : UINT; (*Current mean gray value for third flash color*)
		GrayValue4 : UINT; (*Current mean gray value for fourth flash color*)
		TotalError : ARRAY[1..MAX_NUM_PRODUCTS]OF UINT; (*Total error of mean gray value for all products*)
		LowError : UINT; (*Lowest error found*)
		LowDistance : UINT; (*Distance to next best value*)
		LowIndex : UINT; (*Index of the best value*)
		LowName : STRING[80]; (*Product name of the best value*)
		Status : UINT; (*Status of color detection*)
	END_STRUCT;
END_TYPE

(*-----------------------------------------------------------------------------------------------------------------------------------------*)
(*Image upload structures*)

TYPE
	typVisionImage : 	STRUCT
		CMD : typVisionImageCommand;
		CFG : typVisionImageConfig;
		DAT : typVisionImageData;
	END_STRUCT;
	typVisionImageCommand : 	STRUCT
		CreateDir : BOOL;
		DeleteDir : BOOL;
		DeleteImage : BOOL;
		Refresh : BOOL;
		DownloadImage : BOOL;
		SaveImageOnPLC : BOOL;
		ResetError : BOOL;
		RefreshCrosshair : BOOL;
	END_STRUCT;
	typVisionImageConfig : 	STRUCT
		FileDevice : STRING[80];
		DirName : STRING[80];
		PlkIPWithoutNode : STRING[80];
		EthDevice : STRING[80];
		EthIP : STRING[80];
		ConvertCycles : UDINT;
		Format : USINT; (*0: jpg. 1: bmp*)
		QualityJPG : USINT;
		UploadBmpJpg : BOOL;
		UploadSVG : BOOL;
		MainPageQualityJPG : USINT; (*quality of the jpg image on the main page. min:0, max:100, good value: 30*)
		ImageRotation_deg : UINT; (*rotation of the whole image, steps in degree. Only values 0, 90. 180, 270 make sense*)
	END_STRUCT;
	typVisionImageData : 	STRUCT
		Images : ARRAY[0..19]OF STRING[80];
		Status : UINT;
		VisionDisabled : BOOL;
	END_STRUCT;
END_TYPE

(*-----------------------------------------------------------------------------------------------------------------------------------------*)
(*Vision specific structures*)

TYPE
	typCodeReaderMain : 	STRUCT  (*Code reader structures*)
		CodeType : ARRAY[1..MAX_NUM_RESULTS]OF USINT;
		GradingEnable : BOOL;
		RobustnessEnable : BOOL;
		ParameterMode : USINT;
		ParameterOptimization : USINT;
		BarcodeText : ARRAY[1..MAX_NUM_RESULTS]OF STRING[100];
		BarcodeType : ARRAY[1..MAX_NUM_RESULTS]OF USINT;
		PositionX : ARRAY[1..MAX_NUM_RESULTS]OF DINT;
		PositionY : ARRAY[1..MAX_NUM_RESULTS]OF DINT;
		Orientation : ARRAY[1..MAX_NUM_RESULTS]OF INT;
		Grading : ARRAY[1..MAX_NUM_RESULTS]OF SINT;
		EnhancedGrading : ARRAY[1..23]OF USINT;
	END_STRUCT;
	typBlobMain : 	STRUCT  (*Blob function structures*)
		RegionalFeature : BOOL;
		EnhancedBlobInformation : BOOL := FALSE;
		ModelNumber : ARRAY[1..MAX_NUM_RESULTS]OF USINT;
		Clipped : ARRAY[1..MAX_NUM_RESULTS]OF BOOL;
		Area : ARRAY[1..MAX_NUM_RESULTS]OF UDINT;
		PositionX : ARRAY[1..MAX_NUM_RESULTS]OF DINT;
		PositionY : ARRAY[1..MAX_NUM_RESULTS]OF DINT;
		Orientation : ARRAY[1..MAX_NUM_RESULTS]OF INT;
		MeanGrayValue : ARRAY[1..MAX_NUM_RESULTS]OF USINT;
		Length : ARRAY[1..MAX_NUM_RESULTS]OF UDINT;
		Width : ARRAY[1..MAX_NUM_RESULTS]OF UDINT;
	END_STRUCT;
	typMatchMain : 	STRUCT  (*Match function structures*)
		MinScore : USINT := 70;
		MaxOverlap : USINT;
		ModelNumber : ARRAY[1..MAX_NUM_RESULTS]OF USINT;
		Score : ARRAY[1..MAX_NUM_RESULTS]OF USINT;
		PositionX : ARRAY[1..MAX_NUM_RESULTS]OF DINT;
		PositionY : ARRAY[1..MAX_NUM_RESULTS]OF DINT;
		Orientation : ARRAY[1..MAX_NUM_RESULTS]OF INT;
		Scale : ARRAY[1..MAX_NUM_RESULTS]OF USINT;
		RotCenterX : ARRAY[1..MAX_NUM_RESULTS]OF DINT;
		RotCenterY : ARRAY[1..MAX_NUM_RESULTS]OF DINT;
	END_STRUCT;
	typOCRMain : 	STRUCT  (*OCR function structures*)
		ParameterMode : USINT;
		GradingEnable : BOOL;
		Text : ARRAY[1..MAX_NUM_RESULTS]OF STRING[50];
		Grading : ARRAY[1..MAX_NUM_RESULTS]OF USINT;
		PositionX : ARRAY[1..MAX_NUM_RESULTS]OF DINT;
		PositionY : ARRAY[1..MAX_NUM_RESULTS]OF DINT;
		Orientation : ARRAY[1..MAX_NUM_RESULTS]OF INT;
	END_STRUCT;
	typPixelMain : 	STRUCT  (*OCR function structures*)
		EnhancedPixelCounterInformation : BOOL := FALSE;
		ModelNumber : ARRAY[1..MAX_NUM_RESULTS]OF USINT;
		NumPixels : ARRAY[1..MAX_NUM_RESULTS]OF UDINT;
		MinGray : ARRAY[1..MAX_NUM_RESULTS]OF USINT;
		MaxGray : ARRAY[1..MAX_NUM_RESULTS]OF USINT;
		MeanGray : ARRAY[1..MAX_NUM_RESULTS]OF UINT;
		DeviationGray : ARRAY[1..MAX_NUM_RESULTS]OF UINT;
		MedianGray : ARRAY[1..MAX_NUM_RESULTS]OF USINT;
		ModelArea : ARRAY[1..MAX_NUM_RESULTS]OF UDINT;
		NumConnectedComponents : ARRAY[1..MAX_NUM_RESULTS]OF UINT;
		PositionX : ARRAY[1..MAX_NUM_RESULTS]OF DINT;
		PositionY : ARRAY[1..MAX_NUM_RESULTS]OF DINT;
	END_STRUCT;
	typMTMain : 	STRUCT  (*MT function structures*)
		UseResultAsXY : BOOL;
		ParameterMode : USINT;
		Result : ARRAY[1..MAX_NUM_RESULTS]OF DINT;
	END_STRUCT;
END_TYPE

(*------------------------------------------------------------------------------------------------------------------------------------------------------------------------------------------------------------------------*)
(*Structure that contains the recipe variables*)

TYPE
	recVariable : 	STRUCT
		Cam : ARRAY[1..MAX_NUM_CAMS]OF recVariableCam;
		Light : ARRAY[1..MAX_NUM_LIGHTS]OF recVariableLight;
	END_STRUCT;
	recVariableCam : 	STRUCT
		ApplicationName : STRING[40];
		MaxItemCnt : USINT := 10;
		Timeout : UINT := 5000;
		Gain : USINT;
		Focus : UINT;
		Exposure : UDINT;
		FlashColor : USINT := 1;
		FlashSegment : USINT := 15;
	END_STRUCT;
	recVariableLight : 	STRUCT
		Timeout : UINT := 5000;
		Exposure : UDINT;
		FlashColor : USINT := 1;
		FlashSegment : UINT := 15;
		SetAngle : UINT := 45;
	END_STRUCT;
END_TYPE
```

### VisionVariables.var - not listed in the package file held
```iecst
(*-----------------------------------------------------------------------------------------------------------------------------------------*)
(*Global variables for sensor hardware and vision functions*)
VAR
	gBlob : typBlobMain; (*Data that is specific for the blob function*)
	gCodeReader : typCodeReaderMain; (*Data that is specific for the code reader*)
	gMatch : typMatchMain; (*Data that is specific for the match function*)
	gMT : typMTMain; (*Data that is specific for the measurement function*)
	gOCR : typOCRMain; (*Data that is specific for the OCR function*)
	gPixel : typPixelMain; (*Data that is specific for the Pixel Counter function*)
	gVisionColor : typVisionColor;
	gVisionImage : typVisionImage; (*Data for image handling*)
	gVisionLight : ARRAY[0..MAX_NUM_LIGHTS] OF typLightMain; (*General Light  functions that are independent from the inspection function*)
	gVisionNettime : typVisionNettime; (*Data for nettime calculation*)
	gVisionSensor : ARRAY[0..MAX_NUM_CAMS] OF typVisionMain; (*General vision functions that are independent from the inspection function*)
	gSelectedSensor : UINT := 1; (*Selected camera node number*)
	gSelectedLight : UINT := 1; (*Selected Light node number*)
	NettimeCurrent_us : DINT; (*Current Powerlink nettime*)
END_VAR
VAR RETAIN
	RecipeData : recVariable; (*Structure that contains the recipe variables*)
END_VAR
(*-----------------------------------------------------------------------------------------------------------------------------------------*)
(*Global constants*)
VAR CONSTANT
	MAX_NUM_CAMS : UINT := 6; (*Maximum number of camera's*)
	MAX_NUM_LIGHTS : UINT := 5; (*Maximum number of light's*)
	MAX_NUM_RESULTS : UINT := 10; (*Maximum number of results*)
	MAX_NUM_PRODUCTS : UINT := 8; (*Maximum number of products for color detection*)
	MAX_IDX_VA_LIST : UINT := 19; (*Maximum number of entrys in the Vision Application list*)
	DEVICE_NAME : STRING[40] := 'VisionFileDevice'; (*File device where the images and recipes are stored*)
	NETTIME_DEFAULT_DELAY : UDINT := 30000; (*This delay is used when software trigger is used and nettime is enabled*)
	NETTIME_ENABLE : BOOL := FALSE; (*Enable nettime code, this generates the nettime when using manual triggers*)
	MAX_NUM_CODETYPES : USINT := 69; (*Maximum number of code types*)
END_VAR
VAR
	CodeTypes : {REDUND_UNREPLICABLE} ARRAY[0..MAX_NUM_CODETYPES] OF STRING[80] := ['Auto Identify (0)','2/5 Industrial (1)','2/5 Interleaved (2)','Codebar (3)','Code 32 (4)','Code 39 (5)','Code 93 (6)','Code 128 (7)','MSI (8)','PharmaCode (9)','EAN-8 (10)','EAN-8 Add-On 2 (11)','EAN-8 Add-On 5 (12)','EAN-13 (13)','EAN-13 Add-On 2 (14)','EAN-13 Add-On 5 (15)',4(''),'UPC-A (20)','UPC-A Add-On 2 (21)','UPC-A Add-On 5 (22)','UPC-E (23)','UPC-E Add-On 2 (24)','UPC-E Add-On 5 (25)',4(''),'GS1-128 (30)','GS1 DataBar Omnidirectional (31)','GS1 DataBar Truncated (32)','GS1 DataBar Stacked (33)','GS1 DataBar Stacked Omnidirectional (34)','GS1 DataBar Limited (35)','GS1 DataBar Expanded (36)','GS1 DataBar ExpandedStacked (37)',12(''),'Data Matrix ECC200 (50)','QR Code Model 1 (51)','QR Code Model 2 (52)','Micro QRCode (53)','PDF417 (54)','Aztec Code (55)',4(''),'GS1 Data Matrix (60)','GS1 QR Code Model 1 (61)','GS1 QR Code Model 2 (62)','GS1 Aztec Code (63)',6('')]; (*Codes types for code reading*)
END_VAR
```

### Program Logical/Programs/Vision/Vi_main (IEC)
